LIN {X 0,Y 176.261,Z 619.953,A -85,B 0,C 180,E1 -22409.998,E2 -22409.998} C_VEL
LIN {X 0,Y 176.004,Z 621.002,A -85,B 0,C 180,E1 -22414.579,E2 -22414.579} C_VEL
LIN {X 0,Y 176.334,Z 620.73,A -85,B 0,C 180,E1 -22419.171,E2 -22419.171} C_VEL
LIN {X 0,Y 177.42,Z 619.155,A -85,B 0,C 180,E1 -22423.747,E2 -22423.747} C_VEL
LIN {X 0,Y 179.665,Z 616.268,A -85,B 0,C 180,E1 -22428.234,E2 -22428.234} C_VEL
LIN {X 0,Y 182.692,Z 611.986,A -85,B 0,C 180,E1 -22432.622,E2 -22432.622} C_VEL
LIN {X 0,Y 186.979,Z 606.194,A -85,B 0,C 180,E1 -22436.808,E2 -22436.808} C_VEL
LIN {X 0,Y 191.544,Z 599.723,A -85,B 0,C 180,E1 -22440.296,E2 -22440.296} C_VEL
LIN {X 0,Y 196.849,Z 591.739,A -85,B 0,C 180,E1 -22443.597,E2 -22443.597} C_VEL
LIN {X 0,Y 201.965,Z 583.426,A -85,B 0,C 180,E1 -22446.266,E2 -22446.266} C_VEL
LIN {X 0,Y 207.375,Z 573.579,A -85,B 0,C 180,E1 -22448.786,E2 -22448.786} C_VEL
LIN {X 0,Y 212.33,Z 563.502,A -85,B 0,C 180,E1 -22450.819,E2 -22450.819} C_VEL
LIN {X 0,Y 217.55,Z 551.5,A -85,B 0,C 180,E1 -22452.717,E2 -22452.717} C_VEL
LIN {X 0,Y 221.948,Z 539.683,A -85,B 0,C 180,E1 -22454.155,E2 -22454.155} C_VEL
LIN {X 0,Y 225.975,Z 526.726,A -85,B 0,C 180,E1 -22455.349,E2 -22455.349} C_VEL
LIN {X 0,Y 228.845,Z 514.868,A -85,B 0,C 180,E1 -22456.192,E2 -22456.192} C_VEL
LIN {X 0,Y 231.422,Z 500.809,A -85,B 0,C 180,E1 -22456.897,E2 -22456.897} C_VEL
LIN {X 0,Y 233.066,Z 485.237,A -85,B 0,C 180,E1 -22457.412,E2 -22457.412} C_VEL
LIN {X 0,Y 236.336,Z 441.448,A -85,B 0,C 180,E1 -22458.62,E2 -22458.62} C_VEL
LIN {X 0,Y 231.828,Z 430.629,A -85,B 0,C 180,E1 -22460.893,E2 -22460.893} C_VEL
LIN {X 0,Y 227.529,Z 421.656,A -85,B 0,C 180,E1 -22463.25,E2 -22463.25} C_VEL
LIN {X 0,Y 223.484,Z 413.857,A -85,B 0,C 180,E1 -22465.684,E2 -22465.684} C_VEL
LIN {X 0,Y 219.996,Z 407.651,A -85,B 0,C 180,E1 -22467.999,E2 -22467.999} C_VEL
LIN {X 0,Y 218.272,Z 404.689,A -85,B 0,C 180,E1 -22469.242,E2 -22469.242} C_VEL
LIN {X 0,Y 215.23,Z 399.598,A -85,B 0,C 180,E1 -22471.706,E2 -22471.706} C_VEL
LIN {X 0,Y 211.663,Z 393.98,A -85,B 0,C 180,E1 -22475.117,E2 -22475.117} C_VEL
LIN {X 0,Y 207.412,Z 387.519,A -85,B 0,C 180,E1 -22480.575,E2 -22480.575} C_VEL
LIN {X 0,Y 206.29,Z 386.531,A -85,B 0,C 180,E1 -22482.531,E2 -22482.531} C_VEL
LIN {X 0,Y 204.121,Z 383.562,A -85,B 0,C 180,E1 -22490.763,E2 -22490.763} C_VEL
LIN {X 0,Y 204.159,Z 383.555,A -85,B 0,C 180,E1 -22492.419,E2 -22492.419} C_VEL
LIN {X 0,Y 206.589,Z 386.339,A -85,B 0,C 180,E1 -22500.487,E2 -22500.487} C_VEL
LIN {X 0,Y 207.66,Z 387.333,A -85,B 0,C 180,E1 -22502.289,E2 -22502.289} C_VEL
LIN {X 0,Y 209.529,Z 390.505,A -85,B 0,C 180,E1 -22504.964,E2 -22504.964} C_VEL
LIN {X 0,Y 211.541,Z 392.569,A -85,B 0,C 180,E1 -22507.173,E2 -22507.173} C_VEL
LIN {X 0,Y 213.826,Z 396.048,A -85,B 0,C 180,E1 -22509.458,E2 -22509.458} C_VEL
LIN {X 0,Y 215.381,Z 397.913,A -85,B 0,C 180,E1 -22510.799,E2 -22510.799} C_VEL
LIN {X 0,Y 218.701,Z 402.698,A -85,B 0,C 180,E1 -22513.418,E2 -22513.418} C_VEL
LIN {X 0,Y 222.211,Z 407.786,A -85,B 0,C 180,E1 -22515.784,E2 -22515.784} C_VEL
LIN {X 0,Y 226.377,Z 414.067,A -85,B 0,C 180,E1 -22518.29,E2 -22518.29} C_VEL
LIN {X 0,Y 230.882,Z 421.436,A -85,B 0,C 180,E1 -22520.734,E2 -22520.734} C_VEL
LIN {X 0,Y 235.489,Z 429.755,A -85,B 0,C 180,E1 -22523.009,E2 -22523.009} C_VEL
LIN {X 0,Y 236.939,Z 432.896,A -85,B 0,C 180,E1 -22523.697,E2 -22523.697} C_VEL
LIN {X 0,Y 232.865,Z 484.514,A -85,B 0,C 180,E1 -22525.125,E2 -22525.125} C_VEL
LIN {X 0,Y 230.746,Z 498.985,A -85,B 0,C 180,E1 -22525.793,E2 -22525.793} C_VEL
LIN {X 0,Y 227.765,Z 513.123,A -85,B 0,C 180,E1 -22526.764,E2 -22526.764} C_VEL
LIN {X 0,Y 224.412,Z 525.3,A -85,B 0,C 180,E1 -22527.885,E2 -22527.885} C_VEL
LIN {X 0,Y 220.004,Z 538.449,A -85,B 0,C 180,E1 -22529.488,E2 -22529.488} C_VEL
LIN {X 0,Y 215.564,Z 549.31,A -85,B 0,C 180,E1 -22531.153,E2 -22531.153} C_VEL
LIN {X 0,Y 210.303,Z 560.524,A -85,B 0,C 180,E1 -22533.34,E2 -22533.34} C_VEL
LIN {X 0,Y 205.09,Z 570.271,A -85,B 0,C 180,E1 -22535.761,E2 -22535.761} C_VEL
LIN {X 0,Y 199.851,Z 579.024,A -85,B 0,C 180,E1 -22538.518,E2 -22538.518} C_VEL
LIN {X 0,Y 194.868,Z 586.574,A -85,B 0,C 180,E1 -22541.555,E2 -22541.555} C_VEL
LIN {X 0,Y 189.758,Z 593.653,A -85,B 0,C 180,E1 -22545.279,E2 -22545.279} C_VEL
LIN {X 0,Y 185.363,Z 599.272,A -85,B 0,C 180,E1 -22549.313,E2 -22549.313} C_VEL
LIN {X 0,Y 182.906,Z 602.168,A -85,B 0,C 180,E1 -22552.066,E2 -22552.066} C_VEL
LIN {X 0,Y 181.044,Z 604.278,A -85,B 0,C 180,E1 -22554.606,E2 -22554.606} C_VEL
LIN {X 0,Y 178.48,Z 606.841,A -85,B 0,C 180,E1 -22559.212,E2 -22559.212} C_VEL
LIN {X 0,Y 176.726,Z 607.981,A -85,B 0,C 180,E1 -22564.062,E2 -22564.062} C_VEL
LIN {X 0,Y 176.221,Z 607.996,A -85,B 0,C 180,E1 -22566.529,E2 -22566.529} C_VEL
LIN {X 0,Y 175.676,Z 606.957,A -85,B 0,C 180,E1 -22571.337,E2 -22571.337} C_VEL
LIN {X 0,Y 175.734,Z 605.894,A -85,B 0,C 180,E1 -22573.745,E2 -22573.745} C_VEL
LIN {X 0,Y 176.164,Z 602.698,A -85,B 0,C 180,E1 -22578.496,E2 -22578.496} C_VEL
LIN {X 0,Y 177.143,Z 598.549,A -85,B 0,C 180,E1 -22582.675,E2 -22582.675} C_VEL
LIN {X 0,Y 178.5,Z 593.339,A -85,B 0,C 180,E1 -22586.616,E2 -22586.616} C_VEL
LIN {X 0,Y 180.399,Z 586.664,A -85,B 0,C 180,E1 -22590.56,E2 -22590.56} C_VEL
LIN {X 0,Y 183.061,Z 578.344,A -85,B 0,C 180,E1 -22594.406,E2 -22594.406} C_VEL
LIN {X 0,Y 185.727,Z 569.663,A -85,B 0,C 180,E1 -22597.613,E2 -22597.613} C_VEL
LIN {X 0,Y 188.906,Z 559.128,A -85,B 0,C 180,E1 -22600.722,E2 -22600.722} C_VEL
LIN {X 0,Y 192.339,Z 547.305,A -85,B 0,C 180,E1 -22603.472,E2 -22603.472} C_VEL
LIN {X 0,Y 195.388,Z 535.469,A -85,B 0,C 180,E1 -22605.652,E2 -22605.652} C_VEL
LIN {X 0,Y 198.281,Z 522.429,A -85,B 0,C 180,E1 -22607.536,E2 -22607.536} C_VEL
LIN {X 0,Y 200.684,Z 509.152,A -85,B 0,C 180,E1 -22608.998,E2 -22608.998} C_VEL
LIN {X 0,Y 202.581,Z 494.605,A -85,B 0,C 180,E1 -22610.165,E2 -22610.165} C_VEL
LIN {X 0,Y 203.925,Z 480.192,A -85,B 0,C 180,E1 -22610.907,E2 -22610.907} C_VEL
LIN {X 0,Y 207.782,Z 410.461,A -85,B 0,C 180,E1 -22613.166,E2 -22613.166} C_VEL
LIN {X 0,Y 205.296,Z 404.053,A -85,B 0,C 180,E1 -22613.922,E2 -22613.922} C_VEL
LIN {X 0,Y 197.581,Z 388.625,A -85,B 0,C 180,E1 -22616.238,E2 -22616.238} C_VEL
LIN {X 0,Y 190.271,Z 375.852,A -85,B 0,C 180,E1 -22618.59,E2 -22618.59} C_VEL
LIN {X 0,Y 183.641,Z 365.472,A -85,B 0,C 180,E1 -22620.895,E2 -22620.895} C_VEL
LIN {X 0,Y 181.481,Z 362.093,A -85,B 0,C 180,E1 -22621.698,E2 -22621.698} C_VEL
LIN {X 0,Y 179.169,Z 359.175,A -85,B 0,C 180,E1 -22622.551,E2 -22622.551} C_VEL
LIN {X 0,Y 178.486,Z 356.878,A -85,B 0,C 180,E1 -22622.896,E2 -22622.896} C_VEL
LIN {X 0,Y 178.408,Z 356.871,A -85,B 0,C 180,E1 -22628.016,E2 -22628.016} C_VEL
LIN {X 0,Y 178.394,Z 356.874,A -85,B 0,C 180,E1 -22632.049,E2 -22632.049} C_VEL
LIN {X 0,Y 178.392,Z 356.857,A -85,B 0,C 180,E1 -22635.167,E2 -22635.167} C_VEL
LIN {X 0,Y 178.398,Z 356.885,A -85,B 0,C 180,E1 -22638.463,E2 -22638.463} C_VEL
LIN {X 0,Y 178.42,Z 356.842,A -85,B 0,C 180,E1 -22643.784,E2 -22643.784} C_VEL
LIN {X 0,Y 178.486,Z 356.856,A -85,B 0,C 180,E1 -22646.548,E2 -22646.548} C_VEL
LIN {X 0,Y 178.442,Z 356.873,A -85,B 0,C 180,E1 -22651.796,E2 -22651.796} C_VEL
LIN {X 0,Y 178.508,Z 356.875,A -85,B 0,C 180,E1 -22654.898,E2 -22654.898} C_VEL
LIN {X 0,Y 178.609,Z 356.861,A -85,B 0,C 180,E1 -22661.653,E2 -22661.653} C_VEL
LIN {X 0,Y 178.629,Z 356.813,A -85,B 0,C 180,E1 -22666.346,E2 -22666.346} C_VEL
LIN {X 0,Y 178.908,Z 356.807,A -85,B 0,C 180,E1 -22670.96,E2 -22670.96} C_VEL
LIN {X 0,Y 179.134,Z 356.761,A -85,B 0,C 180,E1 -22677.752,E2 -22677.752} C_VEL
LIN {X 0,Y 179.363,Z 356.721,A -85,B 0,C 180,E1 -22680.001,E2 -22680.001} C_VEL
LIN {X 0,Y 178.848,Z 356.83,A -85,B 0,C 180,E1 -22684.508,E2 -22684.508} C_VEL
LIN {X 0,Y 178.912,Z 356.815,A -85,B 0,C 180,E1 -22689.041,E2 -22689.041} C_VEL
LIN {X 0,Y 178.663,Z 356.846,A -85,B 0,C 180,E1 -22693.653,E2 -22693.653} C_VEL
LIN {X 0,Y 178.63,Z 356.847,A -85,B 0,C 180,E1 -22699.216,E2 -22699.216} C_VEL
LIN {X 0,Y 178.531,Z 356.859,A -85,B 0,C 180,E1 -22705.117,E2 -22705.117} C_VEL
LIN {X 0,Y 178.528,Z 356.862,A -85,B 0,C 180,E1 -22709.993,E2 -22709.993} C_VEL
LIN {X 0,Y 178.49,Z 356.872,A -85,B 0,C 180,E1 -22714.219,E2 -22714.219} C_VEL
LIN {X 0,Y 178.504,Z 356.951,A -85,B 0,C 180,E1 -22718.589,E2 -22718.589} C_VEL
LIN {X 0,Y 179.376,Z 359.579,A -85,B 0,C 180,E1 -22719.002,E2 -22719.002} C_VEL
LIN {X 0,Y 181.535,Z 362.296,A -85,B 0,C 180,E1 -22719.792,E2 -22719.792} C_VEL
LIN {X 0,Y 187.23,Z 372.234,A -85,B 0,C 180,E1 -22721.912,E2 -22721.912} C_VEL
LIN {X 0,Y 193.614,Z 385.014,A -85,B 0,C 180,E1 -22724.147,E2 -22724.147} C_VEL
LIN {X 0,Y 200.31,Z 400.306,A -85,B 0,C 180,E1 -22726.357,E2 -22726.357} C_VEL
LIN {X 0,Y 206.239,Z 416.491,A -85,B 0,C 180,E1 -22728.26,E2 -22728.26} C_VEL
LIN {X 0,Y 207.164,Z 425.712,A -85,B 0,C 180,E1 -22728.83,E2 -22728.83} C_VEL
LIN {X 0,Y 204.565,Z 475.041,A -85,B 0,C 180,E1 -22730.433,E2 -22730.433} C_VEL
LIN {X 0,Y 203.688,Z 480.877,A -85,B 0,C 180,E1 -22730.514,E2 -22730.514} C_VEL
LIN {X 0,Y 197.568,Z 499.736,A -85,B 0,C 180,E1 -22730.355,E2 -22730.355} C_VEL
LIN {X 0,Y 196.339,Z 505.475,A -85,B 0,C 180,E1 -22730.574,E2 -22730.574} C_VEL
LIN {X 0,Y 194.428,Z 518.993,A -85,B 0,C 180,E1 -22731.589,E2 -22731.589} C_VEL
LIN {X 0,Y 191.8,Z 532.414,A -85,B 0,C 180,E1 -22732.963,E2 -22732.963} C_VEL
LIN {X 0,Y 188.72,Z 545.437,A -85,B 0,C 180,E1 -22734.744,E2 -22734.744} C_VEL
LIN {X 0,Y 185.868,Z 556.719,A -85,B 0,C 180,E1 -22736.76,E2 -22736.76} C_VEL
LIN {X 0,Y 183.057,Z 566.038,A -85,B 0,C 180,E1 -22738.78,E2 -22738.78} C_VEL
LIN {X 0,Y 179.87,Z 575.945,A -85,B 0,C 180,E1 -22741.401,E2 -22741.401} C_VEL
LIN {X 0,Y 176.674,Z 585.85,A -85,B 0,C 180,E1 -22744.681,E2 -22744.681} C_VEL
LIN {X 0,Y 173.85,Z 594.782,A -85,B 0,C 180,E1 -22748.404,E2 -22748.404} C_VEL
LIN {X 0,Y 171.762,Z 601.876,A -85,B 0,C 180,E1 -22752.127,E2 -22752.127} C_VEL
LIN {X 0,Y 170.306,Z 607.294,A -85,B 0,C 180,E1 -22755.662,E2 -22755.662} C_VEL
LIN {X 0,Y 169.304,Z 612.981,A -85,B 0,C 180,E1 -22760.44,E2 -22760.44} C_VEL
LIN {X 0,Y 169.089,Z 615.207,A -85,B 0,C 180,E1 -22762.835,E2 -22762.835} C_VEL
LIN {X 0,Y 169.003,Z 617.786,A -85,B 0,C 180,E1 -22766.423,E2 -22766.423} C_VEL
LIN {X 0,Y 169.18,Z 619.597,A -85,B 0,C 180,E1 -22769.998,E2 -22769.998} C_VEL
LIN {X 0,Y 168.926,Z 620.714,A -85,B 0,C 180,E1 -22774.771,E2 -22774.771} C_VEL
LIN {X 0,Y 169.3,Z 620.515,A -85,B 0,C 180,E1 -22779.556,E2 -22779.556} C_VEL
LIN {X 0,Y 170.483,Z 619.019,A -85,B 0,C 180,E1 -22784.318,E2 -22784.318} C_VEL
LIN {X 0,Y 172.88,Z 616.212,A -85,B 0,C 180,E1 -22788.977,E2 -22788.977} C_VEL
LIN {X 0,Y 176.13,Z 612.015,A -85,B 0,C 180,E1 -22793.515,E2 -22793.515} C_VEL
LIN {X 0,Y 180.66,Z 606.311,A -85,B 0,C 180,E1 -22797.826,E2 -22797.826} C_VEL
LIN {X 0,Y 185.457,Z 599.935,A -85,B 0,C 180,E1 -22801.401,E2 -22801.401} C_VEL
LIN {X 0,Y 190.98,Z 592.059,A -85,B 0,C 180,E1 -22804.775,E2 -22804.775} C_VEL
LIN {X 0,Y 196.31,Z 583.865,A -85,B 0,C 180,E1 -22807.486,E2 -22807.486} C_VEL
LIN {X 0,Y 201.755,Z 574.456,A -85,B 0,C 180,E1 -22809.972,E2 -22809.972} C_VEL
LIN {X 0,Y 207.059,Z 564.249,A -85,B 0,C 180,E1 -22812.092,E2 -22812.092} C_VEL
LIN {X 0,Y 212.446,Z 552.457,A -85,B 0,C 180,E1 -22814.001,E2 -22814.001} C_VEL
LIN {X 0,Y 216.969,Z 540.917,A -85,B 0,C 180,E1 -22815.445,E2 -22815.445} C_VEL
LIN {X 0,Y 221.402,Z 527.401,A -85,B 0,C 180,E1 -22816.725,E2 -22816.725} C_VEL
LIN {X 0,Y 224.346,Z 515.777,A -85,B 0,C 180,E1 -22817.57,E2 -22817.57} C_VEL
LIN {X 0,Y 227.127,Z 501.604,A -85,B 0,C 180,E1 -22818.293,E2 -22818.293} C_VEL
LIN {X 0,Y 228.818,Z 486.854,A -85,B 0,C 180,E1 -22818.812,E2 -22818.812} C_VEL
LIN {X 0,Y 232.104,Z 444.116,A -85,B 0,C 180,E1 -22820.001,E2 -22820.001} C_VEL
LIN {X 0,Y 228.046,Z 434.201,A -85,B 0,C 180,E1 -22822.229,E2 -22822.229} C_VEL
LIN {X 0,Y 223.673,Z 424.769,A -85,B 0,C 180,E1 -22824.826,E2 -22824.826} C_VEL
LIN {X 0,Y 218.919,Z 415.596,A -85,B 0,C 180,E1 -22827.982,E2 -22827.982} C_VEL
LIN {X 0,Y 215.795,Z 410.218,A -85,B 0,C 180,E1 -22830.329,E2 -22830.329} C_VEL
LIN {X 0,Y 213.28,Z 405.755,A -85,B 0,C 180,E1 -22832.527,E2 -22832.527} C_VEL
LIN {X 0,Y 209.98,Z 400.378,A -85,B 0,C 180,E1 -22835.876,E2 -22835.876} C_VEL
LIN {X 0,Y 206.116,Z 394.154,A -85,B 0,C 180,E1 -22841.228,E2 -22841.228} C_VEL
LIN {X 0,Y 203.236,Z 390.606,A -85,B 0,C 180,E1 -22850.722,E2 -22850.722} C_VEL
LIN {X 0,Y 203.271,Z 390.593,A -85,B 0,C 180,E1 -22852.385,E2 -22852.385} C_VEL
LIN {X 0,Y 205.888,Z 393.57,A -85,B 0,C 180,E1 -22860.855,E2 -22860.855} C_VEL
LIN {X 0,Y 206.467,Z 394.216,A -85,B 0,C 180,E1 -22861.859,E2 -22861.859} C_VEL
LIN {X 0,Y 208.44,Z 397.561,A -85,B 0,C 180,E1 -22864.786,E2 -22864.786} C_VEL
LIN {X 0,Y 210.08,Z 399.305,A -85,B 0,C 180,E1 -22866.65,E2 -22866.65} C_VEL
LIN {X 0,Y 212.464,Z 402.895,A -85,B 0,C 180,E1 -22869.108,E2 -22869.108} C_VEL
LIN {X 0,Y 213.746,Z 404.582,A -85,B 0,C 180,E1 -22870.264,E2 -22870.264} C_VEL
LIN {X 0,Y 216.777,Z 409.088,A -85,B 0,C 180,E1 -22872.769,E2 -22872.769} C_VEL
LIN {X 0,Y 220.394,Z 414.504,A -85,B 0,C 180,E1 -22875.317,E2 -22875.317} C_VEL
LIN {X 0,Y 224.675,Z 421.287,A -85,B 0,C 180,E1 -22877.977,E2 -22877.977} C_VEL
LIN {X 0,Y 229.43,Z 429.452,A -85,B 0,C 180,E1 -22880.621,E2 -22880.621} C_VEL
LIN {X 0,Y 232.719,Z 435.879,A -85,B 0,C 180,E1 -22882.324,E2 -22882.324} C_VEL
LIN {X 0,Y 228.703,Z 485.113,A -85,B 0,C 180,E1 -22883.709,E2 -22883.709} C_VEL
LIN {X 0,Y 226.642,Z 498.883,A -85,B 0,C 180,E1 -22884.344,E2 -22884.344} C_VEL
LIN {X 0,Y 223.813,Z 512.028,A -85,B 0,C 180,E1 -22885.216,E2 -22885.216} C_VEL
LIN {X 0,Y 219.87,Z 526.017,A -85,B 0,C 180,E1 -22886.496,E2 -22886.496} C_VEL
LIN {X 0,Y 215.74,Z 537.951,A -85,B 0,C 180,E1 -22887.95,E2 -22887.95} C_VEL
LIN {X 0,Y 210.594,Z 550.126,A -85,B 0,C 180,E1 -22889.814,E2 -22889.814} C_VEL
LIN {X 0,Y 205.137,Z 561.245,A -85,B 0,C 180,E1 -22892.016,E2 -22892.016} C_VEL
LIN {X 0,Y 199.943,Z 570.521,A -85,B 0,C 180,E1 -22894.354,E2 -22894.354} C_VEL
LIN {X 0,Y 194.239,Z 579.602,A -85,B 0,C 180,E1 -22897.253,E2 -22897.253} C_VEL
LIN {X 0,Y 189.029,Z 587.098,A -85,B 0,C 180,E1 -22900.347,E2 -22900.347} C_VEL
LIN {X 0,Y 184.35,Z 593.206,A -85,B 0,C 180,E1 -22903.589,E2 -22903.589} C_VEL
LIN {X 0,Y 180.308,Z 598.131,A -85,B 0,C 180,E1 -22906.995,E2 -22906.995} C_VEL
LIN {X 0,Y 176.883,Z 602.005,A -85,B 0,C 180,E1 -22910.53,E2 -22910.53} C_VEL
LIN {X 0,Y 174.427,Z 604.602,A -85,B 0,C 180,E1 -22913.69,E2 -22913.69} C_VEL
LIN {X 0,Y 171.927,Z 606.907,A -85,B 0,C 180,E1 -22917.902,E2 -22917.902} C_VEL
LIN {X 0,Y 169.927,Z 608.23,A -85,B 0,C 180,E1 -22922.941,E2 -22922.941} C_VEL
LIN {X 0,Y 168.883,Z 608.039,A -85,B 0,C 180,E1 -22928.007,E2 -22928.007} C_VEL
LIN {X 0,Y 168.595,Z 606.409,A -85,B 0,C 180,E1 -22933.037,E2 -22933.037} C_VEL
LIN {X 0,Y 168.97,Z 603.345,A -85,B 0,C 180,E1 -22937.999,E2 -22937.999} C_VEL
LIN {X 0,Y 169.743,Z 600.065,A -85,B 0,C 180,E1 -22941.671,E2 -22941.671} C_VEL
LIN {X 0,Y 170.811,Z 595.914,A -85,B 0,C 180,E1 -22945.282,E2 -22945.282} C_VEL
LIN {X 0,Y 172.279,Z 590.738,A -85,B 0,C 180,E1 -22948.833,E2 -22948.833} C_VEL
LIN {X 0,Y 174.641,Z 583.348,A -85,B 0,C 180,E1 -22952.885,E2 -22952.885} C_VEL
LIN {X 0,Y 177.738,Z 574.158,A -85,B 0,C 180,E1 -22956.815,E2 -22956.815} C_VEL
LIN {X 0,Y 180.753,Z 564.552,A -85,B 0,C 180,E1 -22960.079,E2 -22960.079} C_VEL
LIN {X 0,Y 184.07,Z 553.872,A -85,B 0,C 180,E1 -22962.964,E2 -22962.964} C_VEL
LIN {X 0,Y 187.427,Z 542.056,A -85,B 0,C 180,E1 -22965.498,E2 -22965.498} C_VEL
LIN {X 0,Y 190.738,Z 528.898,A -85,B 0,C 180,E1 -22967.699,E2 -22967.699} C_VEL
LIN {X 0,Y 193.347,Z 516.33,A -85,B 0,C 180,E1 -22969.324,E2 -22969.324} C_VEL
LIN {X 0,Y 195.596,Z 502.567,A -85,B 0,C 180,E1 -22970.666,E2 -22970.666} C_VEL
LIN {X 0,Y 197.296,Z 488.463,A -85,B 0,C 180,E1 -22971.618,E2 -22971.618} C_VEL
LIN {X 0,Y 198.522,Z 472.121,A -85,B 0,C 180,E1 -22972.282,E2 -22972.282} C_VEL
LIN {X 0,Y 201.874,Z 411.942,A -85,B 0,C 180,E1 -22974.264,E2 -22974.264} C_VEL
LIN {X 0,Y 196.905,Z 400.974,A -85,B 0,C 180,E1 -22975.814,E2 -22975.814} C_VEL
LIN {X 0,Y 189.681,Z 387.165,A -85,B 0,C 180,E1 -22978.174,E2 -22978.174} C_VEL
LIN {X 0,Y 183.223,Z 376.303,A -85,B 0,C 180,E1 -22980.439,E2 -22980.439} C_VEL
LIN {X 0,Y 179.128,Z 370.041,A -85,B 0,C 180,E1 -22981.961,E2 -22981.961} C_VEL
LIN {X 0,Y 176.415,Z 366.014,A -85,B 0,C 180,E1 -22983.022,E2 -22983.022} C_VEL
LIN {X 0,Y 174.06,Z 362.431,A -85,B 0,C 180,E1 -22983.985,E2 -22983.985} C_VEL
LIN {X 0,Y 172.1,Z 360.028,A -85,B 0,C 180,E1 -22984.785,E2 -22984.785} C_VEL
LIN {X 0,Y 171.39,Z 357.744,A -85,B 0,C 180,E1 -22985.239,E2 -22985.239} C_VEL
LIN {X 0,Y 171.344,Z 357.758,A -85,B 0,C 180,E1 -22988.803,E2 -22988.803} C_VEL
LIN {X 0,Y 171.319,Z 357.735,A -85,B 0,C 180,E1 -22994.22,E2 -22994.22} C_VEL
LIN {X 0,Y 171.331,Z 357.766,A -85,B 0,C 180,E1 -22998.981,E2 -22998.981} C_VEL
LIN {X 0,Y 171.361,Z 357.731,A -85,B 0,C 180,E1 -23002.035,E2 -23002.035} C_VEL
LIN {X 0,Y 171.4,Z 357.719,A -85,B 0,C 180,E1 -23005.095,E2 -23005.095} C_VEL
LIN {X 0,Y 171.41,Z 357.755,A -85,B 0,C 180,E1 -23010.528,E2 -23010.528} C_VEL
LIN {X 0,Y 171.43,Z 357.756,A -85,B 0,C 180,E1 -23015.798,E2 -23015.798} C_VEL
LIN {X 0,Y 171.511,Z 357.745,A -85,B 0,C 180,E1 -23020.865,E2 -23020.865} C_VEL
LIN {X 0,Y 171.545,Z 357.699,A -85,B 0,C 180,E1 -23025.771,E2 -23025.771} C_VEL
LIN {X 0,Y 171.847,Z 357.682,A -85,B 0,C 180,E1 -23030.586,E2 -23030.586} C_VEL
LIN {X 0,Y 171.796,Z 357.702,A -85,B 0,C 180,E1 -23035.308,E2 -23035.308} C_VEL
LIN {X 0,Y 172.327,Z 357.596,A -85,B 0,C 180,E1 -23040.001,E2 -23040.001} C_VEL
LIN {X 0,Y 171.868,Z 357.696,A -85,B 0,C 180,E1 -23047.047,E2 -23047.047} C_VEL
LIN {X 0,Y 171.774,Z 357.713,A -85,B 0,C 180,E1 -23050.897,E2 -23050.897} C_VEL
LIN {X 0,Y 171.56,Z 357.74,A -85,B 0,C 180,E1 -23056.665,E2 -23056.665} C_VEL
LIN {X 0,Y 171.551,Z 357.727,A -85,B 0,C 180,E1 -23059.562,E2 -23059.562} C_VEL
LIN {X 0,Y 171.468,Z 357.739,A -85,B 0,C 180,E1 -23065.611,E2 -23065.611} C_VEL
LIN {X 0,Y 171.446,Z 357.746,A -85,B 0,C 180,E1 -23070.585,E2 -23070.585} C_VEL
LIN {X 0,Y 171.381,Z 357.753,A -85,B 0,C 180,E1 -23076.304,E2 -23076.304} C_VEL
LIN {X 0,Y 172.335,Z 360.479,A -85,B 0,C 180,E1 -23076.797,E2 -23076.797} C_VEL
LIN {X 0,Y 174.274,Z 362.579,A -85,B 0,C 180,E1 -23077.568,E2 -23077.568} C_VEL
LIN {X 0,Y 176.733,Z 366.484,A -85,B 0,C 180,E1 -23078.577,E2 -23078.577} C_VEL
LIN {X 0,Y 181.064,Z 373.766,A -85,B 0,C 180,E1 -23080.28,E2 -23080.28} C_VEL
LIN {X 0,Y 185.126,Z 381.484,A -85,B 0,C 180,E1 -23081.826,E2 -23081.826} C_VEL
LIN {X 0,Y 191.167,Z 394.289,A -85,B 0,C 180,E1 -23084.009,E2 -23084.009} C_VEL
LIN {X 0,Y 196.682,Z 407.982,A -85,B 0,C 180,E1 -23085.925,E2 -23085.925} C_VEL
LIN {X 0,Y 200.633,Z 419.431,A -85,B 0,C 180,E1 -23087.279,E2 -23087.279} C_VEL
LIN {X 0,Y 201.287,Z 426.847,A -85,B 0,C 180,E1 -23087.738,E2 -23087.738} C_VEL
LIN {X 0,Y 197.341,Z 496.005,A -85,B 0,C 180,E1 -23090.067,E2 -23090.067} C_VEL
LIN {X 0,Y 196.339,Z 505.475,A -85,B 0,C 180,E1 -23090.574,E2 -23090.574} C_VEL
LIN {X 0,Y 194.333,Z 513.011,A -85,B 0,C 180,E1 -23090.909,E2 -23090.909} C_VEL
LIN {X 0,Y 187.752,Z 527.343,A -85,B 0,C 180,E1 -23091.486,E2 -23091.486} C_VEL
LIN {X 0,Y 185.679,Z 532.688,A -85,B 0,C 180,E1 -23091.944,E2 -23091.944} C_VEL
LIN {X 0,Y 185.166,Z 534.474,A -85,B 0,C 180,E1 -23092.15,E2 -23092.15} C_VEL
LIN {X 0,Y 182.128,Z 546.755,A -85,B 0,C 180,E1 -23093.949,E2 -23093.949} C_VEL
LIN {X 0,Y 179.392,Z 556.978,A -85,B 0,C 180,E1 -23095.859,E2 -23095.859} C_VEL
LIN {X 0,Y 176.285,Z 566.899,A -85,B 0,C 180,E1 -23098.111,E2 -23098.111} C_VEL
LIN {X 0,Y 172.959,Z 576.61,A -85,B 0,C 180,E1 -23100.814,E2 -23100.814} C_VEL
LIN {X 0,Y 169.711,Z 586.367,A -85,B 0,C 180,E1 -23104.224,E2 -23104.224} C_VEL
LIN {X 0,Y 166.975,Z 594.584,A -85,B 0,C 180,E1 -23107.819,E2 -23107.819} C_VEL
LIN {X 0,Y 164.936,Z 601.113,A -85,B 0,C 180,E1 -23111.36,E2 -23111.36} C_VEL
LIN {X 0,Y 163.379,Z 606.634,A -85,B 0,C 180,E1 -23115.041,E2 -23115.041} C_VEL
LIN {X 0,Y 162.278,Z 612.416,A -85,B 0,C 180,E1 -23120.022,E2 -23120.022} C_VEL
LIN {X 0,Y 161.923,Z 616.563,A -85,B 0,C 180,E1 -23125.018,E2 -23125.018} C_VEL
LIN {X 0,Y 162.081,Z 619.212,A -85,B 0,C 180,E1 -23129.998,E2 -23129.998} C_VEL
LIN {X 0,Y 161.875,Z 620.092,A -85,B 0,C 180,E1 -23133.046,E2 -23133.046} C_VEL
LIN {X 0,Y 161.932,Z 620.52,A -85,B 0,C 180,E1 -23137.479,E2 -23137.479} C_VEL
LIN {X 0,Y 162.792,Z 619.752,A -85,B 0,C 180,E1 -23142.463,E2 -23142.463} C_VEL
LIN {X 0,Y 164.735,Z 617.687,A -85,B 0,C 180,E1 -23147.373,E2 -23147.373} C_VEL
LIN {X 0,Y 167.769,Z 614.279,A -85,B 0,C 180,E1 -23152.147,E2 -23152.147} C_VEL
LIN {X 0,Y 170.735,Z 610.789,A -85,B 0,C 180,E1 -23155.606,E2 -23155.606} C_VEL
LIN {X 0,Y 175.732,Z 604.806,A -85,B 0,C 180,E1 -23159.991,E2 -23159.991} C_VEL
LIN {X 0,Y 181.012,Z 598.127,A -85,B 0,C 180,E1 -23163.589,E2 -23163.589} C_VEL
LIN {X 0,Y 186.994,Z 589.871,A -85,B 0,C 180,E1 -23166.964,E2 -23166.964} C_VEL
LIN {X 0,Y 192.667,Z 581.309,A -85,B 0,C 180,E1 -23169.666,E2 -23169.666} C_VEL
LIN {X 0,Y 198.643,Z 570.995,A -85,B 0,C 180,E1 -23172.236,E2 -23172.236} C_VEL
LIN {X 0,Y 204.606,Z 559.496,A -85,B 0,C 180,E1 -23174.413,E2 -23174.413} C_VEL
LIN {X 0,Y 210.286,Z 546.656,A -85,B 0,C 180,E1 -23176.278,E2 -23176.278} C_VEL
LIN {X 0,Y 215.123,Z 533.815,A -85,B 0,C 180,E1 -23177.656,E2 -23177.656} C_VEL
LIN {X 0,Y 219.033,Z 520.545,A -85,B 0,C 180,E1 -23178.763,E2 -23178.763} C_VEL
LIN {X 0,Y 222.357,Z 506.015,A -85,B 0,C 180,E1 -23179.582,E2 -23179.582} C_VEL
LIN {X 0,Y 224.435,Z 491.745,A -85,B 0,C 180,E1 -23180.152,E2 -23180.152} C_VEL
LIN {X 0,Y 228.089,Z 446.972,A -85,B 0,C 180,E1 -23181.423,E2 -23181.423} C_VEL
LIN {X 0,Y 224.238,Z 437.385,A -85,B 0,C 180,E1 -23183.706,E2 -23183.706} C_VEL
LIN {X 0,Y 220.009,Z 428.358,A -85,B 0,C 180,E1 -23186.412,E2 -23186.412} C_VEL
LIN {X 0,Y 216.252,Z 420.862,A -85,B 0,C 180,E1 -23189.114,E2 -23189.114} C_VEL
LIN {X 0,Y 213.558,Z 415.935,A -85,B 0,C 180,E1 -23191.326,E2 -23191.326} C_VEL
LIN {X 0,Y 211.529,Z 412.129,A -85,B 0,C 180,E1 -23193.216,E2 -23193.216} C_VEL
LIN {X 0,Y 208.465,Z 406.932,A -85,B 0,C 180,E1 -23196.499,E2 -23196.499} C_VEL
LIN {X 0,Y 204.905,Z 400.932,A -85,B 0,C 180,E1 -23201.761,E2 -23201.761} C_VEL
LIN {X 0,Y 202.345,Z 397.667,A -85,B 0,C 180,E1 -23210.681,E2 -23210.681} C_VEL
LIN {X 0,Y 202.372,Z 397.669,A -85,B 0,C 180,E1 -23212.351,E2 -23212.351} C_VEL
LIN {X 0,Y 204.519,Z 400.262,A -85,B 0,C 180,E1 -23219.999,E2 -23219.999} C_VEL
LIN {X 0,Y 205.322,Z 401.215,A -85,B 0,C 180,E1 -23221.501,E2 -23221.501} C_VEL
LIN {X 0,Y 207.195,Z 404.412,A -85,B 0,C 180,E1 -23224.406,E2 -23224.406} C_VEL
LIN {X 0,Y 208.688,Z 406.089,A -85,B 0,C 180,E1 -23226.175,E2 -23226.175} C_VEL
LIN {X 0,Y 211.107,Z 409.755,A -85,B 0,C 180,E1 -23228.752,E2 -23228.752} C_VEL
LIN {X 0,Y 214.459,Z 414.715,A -85,B 0,C 180,E1 -23231.744,E2 -23231.744} C_VEL
LIN {X 0,Y 219.285,Z 422.243,A -85,B 0,C 180,E1 -23235.304,E2 -23235.304} C_VEL
LIN {X 0,Y 224.718,Z 431.483,A -85,B 0,C 180,E1 -23238.684,E2 -23238.684} C_VEL
LIN {X 0,Y 228.68,Z 438.964,A -85,B 0,C 180,E1 -23240.893,E2 -23240.893} C_VEL
LIN {X 0,Y 224.754,Z 485.669,A -85,B 0,C 180,E1 -23242.233,E2 -23242.233} C_VEL
LIN {X 0,Y 222.631,Z 499.216,A -85,B 0,C 180,E1 -23242.853,E2 -23242.853} C_VEL
LIN {X 0,Y 219.404,Z 513.468,A -85,B 0,C 180,E1 -23243.811,E2 -23243.811} C_VEL
LIN {X 0,Y 215.275,Z 527.368,A -85,B 0,C 180,E1 -23245.112,E2 -23245.112} C_VEL
LIN {X 0,Y 211.093,Z 538.81,A -85,B 0,C 180,E1 -23246.527,E2 -23246.527} C_VEL
LIN {X 0,Y 205.661,Z 551.119,A -85,B 0,C 180,E1 -23248.442,E2 -23248.442} C_VEL
LIN {X 0,Y 200.079,Z 561.963,A -85,B 0,C 180,E1 -23250.622,E2 -23250.622} C_VEL
LIN {X 0,Y 194.927,Z 570.766,A -85,B 0,C 180,E1 -23252.873,E2 -23252.873} C_VEL
LIN {X 0,Y 188.818,Z 580.047,A -85,B 0,C 180,E1 -23255.87,E2 -23255.87} C_VEL
LIN {X 0,Y 183.271,Z 587.612,A -85,B 0,C 180,E1 -23259.059,E2 -23259.059} C_VEL
LIN {X 0,Y 177.556,Z 594.598,A -85,B 0,C 180,E1 -23262.964,E2 -23262.964} C_VEL
LIN {X 0,Y 172.805,Z 599.95,A -85,B 0,C 180,E1 -23267.058,E2 -23267.058} C_VEL
LIN {X 0,Y 168.878,Z 603.952,A -85,B 0,C 180,E1 -23271.377,E2 -23271.377} C_VEL
LIN {X 0,Y 165.474,Z 606.958,A -85,B 0,C 180,E1 -23276.489,E2 -23276.489} C_VEL
LIN {X 0,Y 163.17,Z 608.428,A -85,B 0,C 180,E1 -23281.722,E2 -23281.722} C_VEL
LIN {X 0,Y 161.919,Z 608.414,A -85,B 0,C 180,E1 -23287.008,E2 -23287.008} C_VEL
LIN {X 0,Y 161.491,Z 606.918,A -85,B 0,C 180,E1 -23292.266,E2 -23292.266} C_VEL
LIN {X 0,Y 161.559,Z 605.629,A -85,B 0,C 180,E1 -23294.873,E2 -23294.873} C_VEL
LIN {X 0,Y 162.27,Z 601.955,A -85,B 0,C 180,E1 -23300.026,E2 -23300.026} C_VEL
LIN {X 0,Y 163.264,Z 598.092,A -85,B 0,C 180,E1 -23303.927,E2 -23303.927} C_VEL
LIN {X 0,Y 164.559,Z 593.533,A -85,B 0,C 180,E1 -23307.554,E2 -23307.554} C_VEL
LIN {X 0,Y 166.722,Z 586.758,A -85,B 0,C 180,E1 -23311.814,E2 -23311.814} C_VEL
LIN {X 0,Y 169.538,Z 578.638,A -85,B 0,C 180,E1 -23315.802,E2 -23315.802} C_VEL
LIN {X 0,Y 172.592,Z 569.496,A -85,B 0,C 180,E1 -23319.376,E2 -23319.376} C_VEL
LIN {X 0,Y 176.131,Z 558.805,A -85,B 0,C 180,E1 -23322.679,E2 -23322.679} C_VEL
LIN {X 0,Y 179.503,Z 547.994,A -85,B 0,C 180,E1 -23325.326,E2 -23325.326} C_VEL
LIN {X 0,Y 182.832,Z 536.169,A -85,B 0,C 180,E1 -23327.623,E2 -23327.623} C_VEL
LIN {X 0,Y 185.918,Z 523.174,A -85,B 0,C 180,E1 -23329.604,E2 -23329.604} C_VEL
LIN {X 0,Y 188.615,Z 509.378,A -85,B 0,C 180,E1 -23331.19,E2 -23331.19} C_VEL
LIN {X 0,Y 190.592,Z 495.475,A -85,B 0,C 180,E1 -23332.352,E2 -23332.352} C_VEL
LIN {X 0,Y 191.977,Z 481.85,A -85,B 0,C 180,E1 -23333.106,E2 -23333.106} C_VEL
LIN {X 0,Y 196.039,Z 414.514,A -85,B 0,C 180,E1 -23335.379,E2 -23335.379} C_VEL
LIN {X 0,Y 195.436,Z 412.406,A -85,B 0,C 180,E1 -23335.609,E2 -23335.609} C_VEL
LIN {X 0,Y 188.166,Z 397.333,A -85,B 0,C 180,E1 -23338.046,E2 -23338.046} C_VEL
LIN {X 0,Y 181.361,Z 385.035,A -85,B 0,C 180,E1 -23340.497,E2 -23340.497} C_VEL
LIN {X 0,Y 175.189,Z 375.186,A -85,B 0,C 180,E1 -23342.883,E2 -23342.883} C_VEL
LIN {X 0,Y 171.991,Z 370.517,A -85,B 0,C 180,E1 -23344.192,E2 -23344.192} C_VEL
LIN {X 0,Y 170.197,Z 367.779,A -85,B 0,C 180,E1 -23344.966,E2 -23344.966} C_VEL
LIN {X 0,Y 168,Z 364.707,A -85,B 0,C 180,E1 -23345.935,E2 -23345.935} C_VEL
LIN {X 0,Y 167.175,Z 363.442,A -85,B 0,C 180,E1 -23346.317,E2 -23346.317} C_VEL
LIN {X 0,Y 165.255,Z 361.357,A -85,B 0,C 180,E1 -23347.176,E2 -23347.176} C_VEL
LIN {X 0,Y 164.323,Z 358.621,A -85,B 0,C 180,E1 -23347.778,E2 -23347.778} C_VEL
LIN {X 0,Y 164.281,Z 358.614,A -85,B 0,C 180,E1 -23353.344,E2 -23353.344} C_VEL
LIN {X 0,Y 164.261,Z 358.63,A -85,B 0,C 180,E1 -23356.8,E2 -23356.8} C_VEL
LIN {X 0,Y 164.291,Z 358.635,A -85,B 0,C 180,E1 -23360.357,E2 -23360.357} C_VEL
LIN {X 0,Y 164.328,Z 358.594,A -85,B 0,C 180,E1 -23364.353,E2 -23364.353} C_VEL
LIN {X 0,Y 164.373,Z 358.635,A -85,B 0,C 180,E1 -23369.132,E2 -23369.132} C_VEL
LIN {X 0,Y 164.389,Z 358.633,A -85,B 0,C 180,E1 -23374.691,E2 -23374.691} C_VEL
LIN {X 0,Y 164.42,Z 358.624,A -85,B 0,C 180,E1 -23380.119,E2 -23380.119} C_VEL
LIN {X 0,Y 164.475,Z 358.585,A -85,B 0,C 180,E1 -23385.146,E2 -23385.146} C_VEL
LIN {X 0,Y 164.767,Z 358.554,A -85,B 0,C 180,E1 -23390.177,E2 -23390.177} C_VEL
LIN {X 0,Y 164.825,Z 358.575,A -85,B 0,C 180,E1 -23392.652,E2 -23392.652} C_VEL
LIN {X 0,Y 165.29,Z 358.47,A -85,B 0,C 180,E1 -23400.001,E2 -23400.001} C_VEL
LIN {X 0,Y 164.829,Z 358.57,A -85,B 0,C 180,E1 -23407.35,E2 -23407.35} C_VEL
LIN {X 0,Y 164.708,Z 358.593,A -85,B 0,C 180,E1 -23411.06,E2 -23411.06} C_VEL
LIN {X 0,Y 164.49,Z 358.618,A -85,B 0,C 180,E1 -23417.403,E2 -23417.403} C_VEL
LIN {X 0,Y 164.48,Z 358.608,A -85,B 0,C 180,E1 -23419.989,E2 -23419.989} C_VEL
LIN {X 0,Y 164.394,Z 358.622,A -85,B 0,C 180,E1 -23426.13,E2 -23426.13} C_VEL
LIN {X 0,Y 164.384,Z 358.63,A -85,B 0,C 180,E1 -23432.374,E2 -23432.374} C_VEL
LIN {X 0,Y 164.366,Z 358.827,A -85,B 0,C 180,E1 -23433.771,E2 -23433.771} C_VEL
LIN {X 0,Y 165.263,Z 361.329,A -85,B 0,C 180,E1 -23434.287,E2 -23434.287} C_VEL
LIN {X 0,Y 167.323,Z 363.574,A -85,B 0,C 180,E1 -23435.211,E2 -23435.211} C_VEL
LIN {X 0,Y 169.918,Z 367.53,A -85,B 0,C 180,E1 -23436.39,E2 -23436.39} C_VEL
LIN {X 0,Y 171.405,Z 369.637,A -85,B 0,C 180,E1 -23437.03,E2 -23437.03} C_VEL
LIN {X 0,Y 174.72,Z 374.683,A -85,B 0,C 180,E1 -23438.412,E2 -23438.412} C_VEL
LIN {X 0,Y 180.319,Z 385.245,A -85,B 0,C 180,E1 -23440.688,E2 -23440.688} C_VEL
LIN {X 0,Y 186.375,Z 398.383,A -85,B 0,C 180,E1 -23443.021,E2 -23443.021} C_VEL
LIN {X 0,Y 191.688,Z 411.962,A -85,B 0,C 180,E1 -23444.986,E2 -23444.986} C_VEL
LIN {X 0,Y 195.002,Z 421.512,A -85,B 0,C 180,E1 -23446.183,E2 -23446.183} C_VEL
LIN {X 0,Y 195.461,Z 427.757,A -85,B 0,C 180,E1 -23446.57,E2 -23446.57} C_VEL
LIN {X 0,Y 191.441,Z 495.576,A -85,B 0,C 180,E1 -23448.899,E2 -23448.899} C_VEL
LIN {X 0,Y 189.836,Z 509.459,A -85,B 0,C 180,E1 -23449.703,E2 -23449.703} C_VEL
LIN {X 0,Y 187.503,Z 523.711,A -85,B 0,C 180,E1 -23450.935,E2 -23450.935} C_VEL
LIN {X 0,Y 185.166,Z 534.474,A -85,B 0,C 180,E1 -23452.15,E2 -23452.15} C_VEL
LIN {X 0,Y 183.285,Z 539.763,A -85,B 0,C 180,E1 -23452.754,E2 -23452.754} C_VEL
LIN {X 0,Y 178.721,Z 548.035,A -85,B 0,C 180,E1 -23453.657,E2 -23453.657} C_VEL
LIN {X 0,Y 173.943,Z 556.053,A -85,B 0,C 180,E1 -23454.756,E2 -23454.756} C_VEL
LIN {X 0,Y 171.756,Z 560.755,A -85,B 0,C 180,E1 -23455.665,E2 -23455.665} C_VEL
LIN {X 0,Y 168.098,Z 571.736,A -85,B 0,C 180,E1 -23458.49,E2 -23458.49} C_VEL
LIN {X 0,Y 164.332,Z 582.311,A -85,B 0,C 180,E1 -23461.935,E2 -23461.935} C_VEL
LIN {X 0,Y 161.299,Z 591.03,A -85,B 0,C 180,E1 -23465.546,E2 -23465.546} C_VEL
LIN {X 0,Y 158.519,Z 599.324,A -85,B 0,C 180,E1 -23469.901,E2 -23469.901} C_VEL
LIN {X 0,Y 156.477,Z 605.97,A -85,B 0,C 180,E1 -23474.364,E2 -23474.364} C_VEL
LIN {X 0,Y 155.232,Z 611.842,A -85,B 0,C 180,E1 -23479.564,E2 -23479.564} C_VEL
LIN {X 0,Y 154.841,Z 616.077,A -85,B 0,C 180,E1 -23484.789,E2 -23484.789} C_VEL
LIN {X 0,Y 154.986,Z 618.808,A -85,B 0,C 180,E1 -23489.998,E2 -23489.998} C_VEL
LIN {X 0,Y 154.815,Z 619.702,A -85,B 0,C 180,E1 -23492.892,E2 -23492.892} C_VEL
LIN {X 0,Y 154.887,Z 620.238,A -85,B 0,C 180,E1 -23497.821,E2 -23497.821} C_VEL
LIN {X 0,Y 155.828,Z 619.553,A -85,B 0,C 180,E1 -23503.03,E2 -23503.03} C_VEL
LIN {X 0,Y 157.93,Z 617.577,A -85,B 0,C 180,E1 -23508.147,E2 -23508.147} C_VEL
LIN {X 0,Y 161.157,Z 614.263,A -85,B 0,C 180,E1 -23513.107,E2 -23513.107} C_VEL
LIN {X 0,Y 165.546,Z 609.504,A -85,B 0,C 180,E1 -23517.836,E2 -23517.836} C_VEL
LIN {X 0,Y 171.083,Z 603.172,A -85,B 0,C 180,E1 -23522.276,E2 -23522.276} C_VEL
LIN {X 0,Y 176.803,Z 596.175,A -85,B 0,C 180,E1 -23525.893,E2 -23525.893} C_VEL
LIN {X 0,Y 183.296,Z 587.551,A -85,B 0,C 180,E1 -23529.243,E2 -23529.243} C_VEL
LIN {X 0,Y 189.253,Z 578.601,A -85,B 0,C 180,E1 -23531.944,E2 -23531.944} C_VEL
LIN {X 0,Y 194.572,Z 569.757,A -85,B 0,C 180,E1 -23534.049,E2 -23534.049} C_VEL
LIN {X 0,Y 200.815,Z 558.089,A -85,B 0,C 180,E1 -23536.202,E2 -23536.202} C_VEL
LIN {X 0,Y 206.111,Z 546.448,A -85,B 0,C 180,E1 -23537.868,E2 -23537.868} C_VEL
LIN {X 0,Y 211.09,Z 533.631,A -85,B 0,C 180,E1 -23539.235,E2 -23539.235} C_VEL
LIN {X 0,Y 215.125,Z 520.383,A -85,B 0,C 180,E1 -23540.33,E2 -23540.33} C_VEL
LIN {X 0,Y 218.484,Z 506.193,A -85,B 0,C 180,E1 -23541.128,E2 -23541.128} C_VEL
LIN {X 0,Y 220.687,Z 491.622,A -85,B 0,C 180,E1 -23541.709,E2 -23541.709} C_VEL
LIN {X 0,Y 224.23,Z 449.931,A -85,B 0,C 180,E1 -23542.887,E2 -23542.887} C_VEL
LIN {X 0,Y 220.244,Z 439.918,A -85,B 0,C 180,E1 -23545.449,E2 -23545.449} C_VEL
LIN {X 0,Y 216.153,Z 431.103,A -85,B 0,C 180,E1 -23548.331,E2 -23548.331} C_VEL
LIN {X 0,Y 213.068,Z 424.742,A -85,B 0,C 180,E1 -23550.835,E2 -23550.835} C_VEL
LIN {X 0,Y 209.77,Z 418.467,A -85,B 0,C 180,E1 -23553.954,E2 -23553.954} C_VEL
LIN {X 0,Y 206.911,Z 413.411,A -85,B 0,C 180,E1 -23557.207,E2 -23557.207} C_VEL
LIN {X 0,Y 203.902,Z 407.945,A -85,B 0,C 180,E1 -23561.928,E2 -23561.928} C_VEL
LIN {X 0,Y 201.452,Z 404.733,A -85,B 0,C 180,E1 -23570.639,E2 -23570.639} C_VEL
LIN {X 0,Y 201.474,Z 404.731,A -85,B 0,C 180,E1 -23572.317,E2 -23572.317} C_VEL
LIN {X 0,Y 203.808,Z 407.502,A -85,B 0,C 180,E1 -23580.376,E2 -23580.376} C_VEL
LIN {X 0,Y 204.517,Z 408.946,A -85,B 0,C 180,E1 -23581.784,E2 -23581.784} C_VEL
LIN {X 0,Y 207.336,Z 412.971,A -85,B 0,C 180,E1 -23585.733,E2 -23585.733} C_VEL
LIN {X 0,Y 210.358,Z 417.576,A -85,B 0,C 180,E1 -23588.992,E2 -23588.992} C_VEL
LIN {X 0,Y 213.54,Z 422.721,A -85,B 0,C 180,E1 -23591.859,E2 -23591.859} C_VEL
LIN {X 0,Y 217.13,Z 428.471,A -85,B 0,C 180,E1 -23594.588,E2 -23594.588} C_VEL
LIN {X 0,Y 222.247,Z 437.469,A -85,B 0,C 180,E1 -23597.926,E2 -23597.926} C_VEL
LIN {X 0,Y 224.807,Z 442.391,A -85,B 0,C 180,E1 -23599.442,E2 -23599.442} C_VEL
LIN {X 0,Y 221.046,Z 485.613,A -85,B 0,C 180,E1 -23600.676,E2 -23600.676} C_VEL
LIN {X 0,Y 218.951,Z 498.807,A -85,B 0,C 180,E1 -23601.263,E2 -23601.263} C_VEL
LIN {X 0,Y 215.802,Z 512.608,A -85,B 0,C 180,E1 -23602.168,E2 -23602.168} C_VEL
LIN {X 0,Y 212.01,Z 525.322,A -85,B 0,C 180,E1 -23603.304,E2 -23603.304} C_VEL
LIN {X 0,Y 207.203,Z 538.37,A -85,B 0,C 180,E1 -23604.868,E2 -23604.868} C_VEL
LIN {X 0,Y 201.7,Z 550.476,A -85,B 0,C 180,E1 -23606.712,E2 -23606.712} C_VEL
LIN {X 0,Y 195.746,Z 561.704,A -85,B 0,C 180,E1 -23608.942,E2 -23608.942} C_VEL
LIN {X 0,Y 189.593,Z 571.741,A -85,B 0,C 180,E1 -23611.511,E2 -23611.511} C_VEL
LIN {X 0,Y 183.326,Z 580.725,A -85,B 0,C 180,E1 -23614.494,E2 -23614.494} C_VEL
LIN {X 0,Y 177.6,Z 588.115,A -85,B 0,C 180,E1 -23617.683,E2 -23617.683} C_VEL
LIN {X 0,Y 172.079,Z 594.551,A -85,B 0,C 180,E1 -23621.332,E2 -23621.332} C_VEL
LIN {X 0,Y 166.684,Z 600.265,A -85,B 0,C 180,E1 -23625.788,E2 -23625.788} C_VEL
LIN {X 0,Y 162.924,Z 603.862,A -85,B 0,C 180,E1 -23629.684,E2 -23629.684} C_VEL
LIN {X 0,Y 160.882,Z 605.634,A -85,B 0,C 180,E1 -23632.299,E2 -23632.299} C_VEL
LIN {X 0,Y 157.692,Z 607.998,A -85,B 0,C 180,E1 -23637.672,E2 -23637.672} C_VEL
LIN {X 0,Y 155.615,Z 608.858,A -85,B 0,C 180,E1 -23643.155,E2 -23643.155} C_VEL
LIN {X 0,Y 155.001,Z 608.737,A -85,B 0,C 180,E1 -23645.919,E2 -23645.919} C_VEL
LIN {X 0,Y 154.412,Z 607.414,A -85,B 0,C 180,E1 -23651.424,E2 -23651.424} C_VEL
LIN {X 0,Y 154.439,Z 606.201,A -85,B 0,C 180,E1 -23654.157,E2 -23654.157} C_VEL
LIN {X 0,Y 155.066,Z 602.657,A -85,B 0,C 180,E1 -23659.558,E2 -23659.558} C_VEL
LIN {X 0,Y 156.118,Z 598.694,A -85,B 0,C 180,E1 -23663.857,E2 -23663.857} C_VEL
LIN {X 0,Y 157.889,Z 592.707,A -85,B 0,C 180,E1 -23668.727,E2 -23668.727} C_VEL
LIN {X 0,Y 160.31,Z 585.643,A -85,B 0,C 180,E1 -23673.144,E2 -23673.144} C_VEL
LIN {X 0,Y 163.481,Z 576.886,A -85,B 0,C 180,E1 -23677.412,E2 -23677.412} C_VEL
LIN {X 0,Y 166.706,Z 567.743,A -85,B 0,C 180,E1 -23680.938,E2 -23680.938} C_VEL
LIN {X 0,Y 170.48,Z 556.661,A -85,B 0,C 180,E1 -23684.323,E2 -23684.323} C_VEL
LIN {X 0,Y 174.054,Z 545.338,A -85,B 0,C 180,E1 -23687.024,E2 -23687.024} C_VEL
LIN {X 0,Y 177.613,Z 532.774,A -85,B 0,C 180,E1 -23689.355,E2 -23689.355} C_VEL
LIN {X 0,Y 180.459,Z 520.794,A -85,B 0,C 180,E1 -23691.102,E2 -23691.102} C_VEL
LIN {X 0,Y 182.995,Z 507.481,A -85,B 0,C 180,E1 -23692.587,E2 -23692.587} C_VEL
LIN {X 0,Y 185.043,Z 493.202,A -85,B 0,C 180,E1 -23693.727,E2 -23693.727} C_VEL
LIN {X 0,Y 186.352,Z 479.506,A -85,B 0,C 180,E1 -23694.438,E2 -23694.438} C_VEL
LIN {X 0,Y 190.32,Z 416.188,A -85,B 0,C 180,E1 -23696.596,E2 -23696.596} C_VEL
LIN {X 0,Y 184.958,Z 404.526,A -85,B 0,C 180,E1 -23698.499,E2 -23698.499} C_VEL
LIN {X 0,Y 178.391,Z 392.102,A -85,B 0,C 180,E1 -23700.966,E2 -23700.966} C_VEL
LIN {X 0,Y 171.513,Z 380.706,A -85,B 0,C 180,E1 -23703.743,E2 -23703.743} C_VEL
LIN {X 0,Y 166.038,Z 372.612,A -85,B 0,C 180,E1 -23706.15,E2 -23706.15} C_VEL
LIN {X 0,Y 163.557,Z 369.022,A -85,B 0,C 180,E1 -23707.327,E2 -23707.327} C_VEL
LIN {X 0,Y 161.167,Z 365.821,A -85,B 0,C 180,E1 -23708.504,E2 -23708.504} C_VEL
LIN {X 0,Y 160.473,Z 364.616,A -85,B 0,C 180,E1 -23708.877,E2 -23708.877} C_VEL
LIN {X 0,Y 158.255,Z 362.404,A -85,B 0,C 180,E1 -23709.993,E2 -23709.993} C_VEL
LIN {X 0,Y 157.315,Z 360.096,A -85,B 0,C 180,E1 -23710.584,E2 -23710.584} C_VEL
LIN {X 0,Y 157.209,Z 359.526,A -85,B 0,C 180,E1 -23710.769,E2 -23710.769} C_VEL
LIN {X 0,Y 157.179,Z 359.498,A -85,B 0,C 180,E1 -23715.68,E2 -23715.68} C_VEL
LIN {X 0,Y 157.199,Z 359.502,A -85,B 0,C 180,E1 -23721.252,E2 -23721.252} C_VEL
LIN {X 0,Y 157.276,Z 359.471,A -85,B 0,C 180,E1 -23724.486,E2 -23724.486} C_VEL
LIN {X 0,Y 157.286,Z 359.512,A -85,B 0,C 180,E1 -23728.104,E2 -23728.104} C_VEL
LIN {X 0,Y 157.313,Z 359.506,A -85,B 0,C 180,E1 -23733.466,E2 -23733.466} C_VEL
LIN {X 0,Y 157.363,Z 359.501,A -85,B 0,C 180,E1 -23739.704,E2 -23739.704} C_VEL
LIN {X 0,Y 157.409,Z 359.473,A -85,B 0,C 180,E1 -23744.462,E2 -23744.462} C_VEL
LIN {X 0,Y 157.69,Z 359.426,A -85,B 0,C 180,E1 -23749.732,E2 -23749.732} C_VEL
LIN {X 0,Y 157.763,Z 359.452,A -85,B 0,C 180,E1 -23752.321,E2 -23752.321} C_VEL
LIN {X 0,Y 158.251,Z 359.345,A -85,B 0,C 180,E1 -23760.001,E2 -23760.001} C_VEL
LIN {X 0,Y 157.767,Z 359.448,A -85,B 0,C 180,E1 -23767.681,E2 -23767.681} C_VEL
LIN {X 0,Y 157.643,Z 359.474,A -85,B 0,C 180,E1 -23771.236,E2 -23771.236} C_VEL
LIN {X 0,Y 157.448,Z 359.494,A -85,B 0,C 180,E1 -23775.536,E2 -23775.536} C_VEL
LIN {X 0,Y 157.376,Z 359.497,A -85,B 0,C 180,E1 -23780.933,E2 -23780.933} C_VEL
LIN {X 0,Y 157.317,Z 359.507,A -85,B 0,C 180,E1 -23786.681,E2 -23786.681} C_VEL
LIN {X 0,Y 157.35,Z 359.502,A -85,B 0,C 180,E1 -23790.815,E2 -23790.815} C_VEL
LIN {X 0,Y 158.293,Z 362.292,A -85,B 0,C 180,E1 -23791.478,E2 -23791.478} C_VEL
LIN {X 0,Y 160.348,Z 364.468,A -85,B 0,C 180,E1 -23792.522,E2 -23792.522} C_VEL
LIN {X 0,Y 161.087,Z 365.625,A -85,B 0,C 180,E1 -23792.91,E2 -23792.91} C_VEL
LIN {X 0,Y 163.312,Z 368.73,A -85,B 0,C 180,E1 -23794.018,E2 -23794.018} C_VEL
LIN {X 0,Y 167.643,Z 374.956,A -85,B 0,C 180,E1 -23796.043,E2 -23796.043} C_VEL
LIN {X 0,Y 170.834,Z 379.921,A -85,B 0,C 180,E1 -23797.452,E2 -23797.452} C_VEL
LIN {X 0,Y 176.06,Z 390.059,A -85,B 0,C 180,E1 -23799.695,E2 -23799.695} C_VEL
LIN {X 0,Y 181.786,Z 402.857,A -85,B 0,C 180,E1 -23802.04,E2 -23802.04} C_VEL
LIN {X 0,Y 187.354,Z 417.504,A -85,B 0,C 180,E1 -23804.223,E2 -23804.223} C_VEL
LIN {X 0,Y 189.497,Z 424.522,A -85,B 0,C 180,E1 -23805.079,E2 -23805.079} C_VEL
LIN {X 0,Y 189.697,Z 429.407,A -85,B 0,C 180,E1 -23805.361,E2 -23805.361} C_VEL
LIN {X 0,Y 185.597,Z 495.447,A -85,B 0,C 180,E1 -23807.674,E2 -23807.674} C_VEL
LIN {X 0,Y 183.945,Z 509.29,A -85,B 0,C 180,E1 -23808.495,E2 -23808.495} C_VEL
LIN {X 0,Y 181.531,Z 523.52,A -85,B 0,C 180,E1 -23809.753,E2 -23809.753} C_VEL
LIN {X 0,Y 178.527,Z 536.665,A -85,B 0,C 180,E1 -23811.32,E2 -23811.32} C_VEL
LIN {X 0,Y 175.576,Z 547.992,A -85,B 0,C 180,E1 -23813.098,E2 -23813.098} C_VEL
LIN {X 0,Y 173.043,Z 556.951,A -85,B 0,C 180,E1 -23814.832,E2 -23814.832} C_VEL
LIN {X 0,Y 171.756,Z 560.755,A -85,B 0,C 180,E1 -23815.665,E2 -23815.665} C_VEL
LIN {X 0,Y 169.506,Z 565.395,A -85,B 0,C 180,E1 -23816.646,E2 -23816.646} C_VEL
LIN {X 0,Y 164.394,Z 572.592,A -85,B 0,C 180,E1 -23818.208,E2 -23818.208} C_VEL
LIN {X 0,Y 159.366,Z 579.322,A -85,B 0,C 180,E1 -23820.058,E2 -23820.058} C_VEL
LIN {X 0,Y 157.294,Z 583.224,A -85,B 0,C 180,E1 -23821.473,E2 -23821.473} C_VEL
LIN {X 0,Y 154.301,Z 591.423,A -85,B 0,C 180,E1 -23825.08,E2 -23825.08} C_VEL
LIN {X 0,Y 151.791,Z 598.556,A -85,B 0,C 180,E1 -23828.969,E2 -23828.969} C_VEL
LIN {X 0,Y 149.607,Z 605.306,A -85,B 0,C 180,E1 -23833.626,E2 -23833.626} C_VEL
LIN {X 0,Y 148.213,Z 611.269,A -85,B 0,C 180,E1 -23839.064,E2 -23839.064} C_VEL
LIN {X 0,Y 147.887,Z 613.626,A -85,B 0,C 180,E1 -23841.801,E2 -23841.801} C_VEL
LIN {X 0,Y 147.744,Z 615.59,A -85,B 0,C 180,E1 -23844.538,E2 -23844.538} C_VEL
LIN {X 0,Y 147.758,Z 617.178,A -85,B 0,C 180,E1 -23847.271,E2 -23847.271} C_VEL
LIN {X 0,Y 147.893,Z 618.403,A -85,B 0,C 180,E1 -23849.998,E2 -23849.998} C_VEL
LIN {X 0,Y 147.757,Z 619.255,A -85,B 0,C 180,E1 -23852.724,E2 -23852.724} C_VEL
LIN {X 0,Y 147.837,Z 619.948,A -85,B 0,C 180,E1 -23858.197,E2 -23858.197} C_VEL
LIN {X 0,Y 148.889,Z 619.34,A -85,B 0,C 180,E1 -23863.649,E2 -23863.649} C_VEL
LIN {X 0,Y 151.16,Z 617.443,A -85,B 0,C 180,E1 -23868.991,E2 -23868.991} C_VEL
LIN {X 0,Y 154.602,Z 614.221,A -85,B 0,C 180,E1 -23874.147,E2 -23874.147} C_VEL
LIN {X 0,Y 159.281,Z 609.575,A -85,B 0,C 180,E1 -23879.033,E2 -23879.033} C_VEL
LIN {X 0,Y 165.125,Z 603.336,A -85,B 0,C 180,E1 -23883.591,E2 -23883.591} C_VEL
LIN {X 0,Y 171.095,Z 596.461,A -85,B 0,C 180,E1 -23887.289,E2 -23887.289} C_VEL
LIN {X 0,Y 177.879,Z 587.976,A -85,B 0,C 180,E1 -23890.683,E2 -23890.683} C_VEL
LIN {X 0,Y 184.066,Z 579.18,A -85,B 0,C 180,E1 -23893.412,E2 -23893.412} C_VEL
LIN {X 0,Y 190.757,Z 568.564,A -85,B 0,C 180,E1 -23895.922,E2 -23895.922} C_VEL
LIN {X 0,Y 196.625,Z 557.876,A -85,B 0,C 180,E1 -23897.871,E2 -23897.871} C_VEL
LIN {X 0,Y 202.099,Z 546.247,A -85,B 0,C 180,E1 -23899.523,E2 -23899.523} C_VEL
LIN {X 0,Y 207.228,Z 533.445,A -85,B 0,C 180,E1 -23900.873,E2 -23900.873} C_VEL
LIN {X 0,Y 211.384,Z 520.221,A -85,B 0,C 180,E1 -23901.954,E2 -23901.954} C_VEL
LIN {X 0,Y 214.925,Z 505.623,A -85,B 0,C 180,E1 -23902.756,E2 -23902.756} C_VEL
LIN {X 0,Y 217.096,Z 491.71,A -85,B 0,C 180,E1 -23903.307,E2 -23903.307} C_VEL
LIN {X 0,Y 220.551,Z 452.956,A -85,B 0,C 180,E1 -23904.382,E2 -23904.382} C_VEL
LIN {X 0,Y 216.957,Z 443.926,A -85,B 0,C 180,E1 -23906.871,E2 -23906.871} C_VEL
LIN {X 0,Y 213.289,Z 435.687,A -85,B 0,C 180,E1 -23909.691,E2 -23909.691} C_VEL
LIN {X 0,Y 210.287,Z 429.295,A -85,B 0,C 180,E1 -23912.397,E2 -23912.397} C_VEL
LIN {X 0,Y 207.901,Z 424.492,A -85,B 0,C 180,E1 -23914.869,E2 -23914.869} C_VEL
LIN {X 0,Y 205.331,Z 419.767,A -85,B 0,C 180,E1 -23918.007,E2 -23918.007} C_VEL
LIN {X 0,Y 202.762,Z 414.809,A -85,B 0,C 180,E1 -23922.368,E2 -23922.368} C_VEL
LIN {X 0,Y 200.562,Z 411.782,A -85,B 0,C 180,E1 -23930.597,E2 -23930.597} C_VEL
LIN {X 0,Y 200.577,Z 411.791,A -85,B 0,C 180,E1 -23932.282,E2 -23932.282} C_VEL
LIN {X 0,Y 202.704,Z 414.418,A -85,B 0,C 180,E1 -23939.999,E2 -23939.999} C_VEL
LIN {X 0,Y 205.353,Z 418.801,A -85,B 0,C 180,E1 -23944.445,E2 -23944.445} C_VEL
LIN {X 0,Y 206.533,Z 420.852,A -85,B 0,C 180,E1 -23945.965,E2 -23945.965} C_VEL
LIN {X 0,Y 208.859,Z 424.334,A -85,B 0,C 180,E1 -23948.499,E2 -23948.499} C_VEL
LIN {X 0,Y 212.29,Z 430.02,A -85,B 0,C 180,E1 -23951.683,E2 -23951.683} C_VEL
LIN {X 0,Y 216.033,Z 436.497,A -85,B 0,C 180,E1 -23954.6,E2 -23954.6} C_VEL
LIN {X 0,Y 220.227,Z 444.296,A -85,B 0,C 180,E1 -23957.417,E2 -23957.417} C_VEL
LIN {X 0,Y 221.038,Z 445.892,A -85,B 0,C 180,E1 -23957.926,E2 -23957.926} C_VEL
LIN {X 0,Y 217.463,Z 485.893,A -85,B 0,C 180,E1 -23959.082,E2 -23959.082} C_VEL
LIN {X 0,Y 215.266,Z 499.24,A -85,B 0,C 180,E1 -23959.669,E2 -23959.669} C_VEL
LIN {X 0,Y 212.037,Z 512.939,A -85,B 0,C 180,E1 -23960.559,E2 -23960.559} C_VEL
LIN {X 0,Y 208.056,Z 525.838,A -85,B 0,C 180,E1 -23961.705,E2 -23961.705} C_VEL
LIN {X 0,Y 203.46,Z 537.909,A -85,B 0,C 180,E1 -23963.125,E2 -23963.125} C_VEL
LIN {X 0,Y 197.935,Z 549.785,A -85,B 0,C 180,E1 -23964.891,E2 -23964.891} C_VEL
LIN {X 0,Y 192.172,Z 560.442,A -85,B 0,C 180,E1 -23966.952,E2 -23966.952} C_VEL
LIN {X 0,Y 185.703,Z 570.734,A -85,B 0,C 180,E1 -23969.495,E2 -23969.495} C_VEL
LIN {X 0,Y 179.107,Z 579.964,A -85,B 0,C 180,E1 -23972.478,E2 -23972.478} C_VEL
LIN {X 0,Y 172.06,Z 588.639,A -85,B 0,C 180,E1 -23976.228,E2 -23976.228} C_VEL
LIN {X 0,Y 165.779,Z 595.473,A -85,B 0,C 180,E1 -23980.267,E2 -23980.267} C_VEL
LIN {X 0,Y 160.61,Z 600.6,A -85,B 0,C 180,E1 -23984.436,E2 -23984.436} C_VEL
LIN {X 0,Y 157.151,Z 603.738,A -85,B 0,C 180,E1 -23987.873,E2 -23987.873} C_VEL
LIN {X 0,Y 154.868,Z 605.612,A -85,B 0,C 180,E1 -23990.559,E2 -23990.559} C_VEL
LIN {X 0,Y 151.258,Z 608.117,A -85,B 0,C 180,E1 -23996.116,E2 -23996.116} C_VEL
LIN {X 0,Y 148.881,Z 609.109,A -85,B 0,C 180,E1 -24001.835,E2 -24001.835} C_VEL
LIN {X 0,Y 148.139,Z 609.053,A -85,B 0,C 180,E1 -24004.727,E2 -24004.727} C_VEL
LIN {X 0,Y 147.325,Z 607.863,A -85,B 0,C 180,E1 -24010.495,E2 -24010.495} C_VEL
LIN {X 0,Y 147.316,Z 606.727,A -85,B 0,C 180,E1 -24013.37,E2 -24013.37} C_VEL
LIN {X 0,Y 147.853,Z 603.36,A -85,B 0,C 180,E1 -24019.042,E2 -24019.042} C_VEL
LIN {X 0,Y 148.715,Z 600.072,A -85,B 0,C 180,E1 -24022.933,E2 -24022.933} C_VEL
LIN {X 0,Y 150.147,Z 595.352,A -85,B 0,C 180,E1 -24027.32,E2 -24027.32} C_VEL
LIN {X 0,Y 152.321,Z 588.899,A -85,B 0,C 180,E1 -24031.985,E2 -24031.985} C_VEL
LIN {X 0,Y 155.331,Z 581.012,A -85,B 0,C 180,E1 -24036.414,E2 -24036.414} C_VEL
LIN {X 0,Y 158.508,Z 572.462,A -85,B 0,C 180,E1 -24040.218,E2 -24040.218} C_VEL
LIN {X 0,Y 162.199,Z 562.345,A -85,B 0,C 180,E1 -24043.789,E2 -24043.789} C_VEL
LIN {X 0,Y 166.183,Z 551.007,A -85,B 0,C 180,E1 -24046.905,E2 -24046.905} C_VEL
LIN {X 0,Y 169.649,Z 539.738,A -85,B 0,C 180,E1 -24049.357,E2 -24049.357} C_VEL
LIN {X 0,Y 172.996,Z 527.433,A -85,B 0,C 180,E1 -24051.448,E2 -24051.448} C_VEL
LIN {X 0,Y 175.854,Z 514.763,A -85,B 0,C 180,E1 -24053.112,E2 -24053.112} C_VEL
LIN {X 0,Y 178.311,Z 500.309,A -85,B 0,C 180,E1 -24054.527,E2 -24054.527} C_VEL
LIN {X 0,Y 180.144,Z 485.809,A -85,B 0,C 180,E1 -24055.466,E2 -24055.466} C_VEL
LIN {X 0,Y 182.152,Z 457.345,A -85,B 0,C 180,E1 -24056.527,E2 -24056.527} C_VEL
LIN {X 0,Y 184.582,Z 418.003,A -85,B 0,C 180,E1 -24057.909,E2 -24057.909} C_VEL
LIN {X 0,Y 177.361,Z 402.81,A -85,B 0,C 180,E1 -24060.678,E2 -24060.678} C_VEL
LIN {X 0,Y 170.949,Z 391.344,A -85,B 0,C 180,E1 -24063.296,E2 -24063.296} C_VEL
LIN {X 0,Y 164.812,Z 381.536,A -85,B 0,C 180,E1 -24066.029,E2 -24066.029} C_VEL
LIN {X 0,Y 160.003,Z 374.485,A -85,B 0,C 180,E1 -24068.385,E2 -24068.385} C_VEL
LIN {X 0,Y 157.446,Z 370.792,A -85,B 0,C 180,E1 -24069.742,E2 -24069.742} C_VEL
LIN {X 0,Y 154.551,Z 367.275,A -85,B 0,C 180,E1 -24071.328,E2 -24071.328} C_VEL
LIN {X 0,Y 153.565,Z 365.618,A -85,B 0,C 180,E1 -24071.927,E2 -24071.927} C_VEL
LIN {X 0,Y 151.282,Z 363.489,A -85,B 0,C 180,E1 -24073.24,E2 -24073.24} C_VEL
LIN {X 0,Y 150.269,Z 361.14,A -85,B 0,C 180,E1 -24073.965,E2 -24073.965} C_VEL
LIN {X 0,Y 150.124,Z 360.371,A -85,B 0,C 180,E1 -24074.112,E2 -24074.112} C_VEL
LIN {X 0,Y 150.139,Z 360.406,A -85,B 0,C 180,E1 -24079.056,E2 -24079.056} C_VEL
LIN {X 0,Y 150.178,Z 360.357,A -85,B 0,C 180,E1 -24082.712,E2 -24082.712} C_VEL
LIN {X 0,Y 150.211,Z 360.382,A -85,B 0,C 180,E1 -24087.374,E2 -24087.374} C_VEL
LIN {X 0,Y 150.231,Z 360.384,A -85,B 0,C 180,E1 -24092.732,E2 -24092.732} C_VEL
LIN {X 0,Y 150.287,Z 360.379,A -85,B 0,C 180,E1 -24099.279,E2 -24099.279} C_VEL
LIN {X 0,Y 150.315,Z 360.367,A -85,B 0,C 180,E1 -24103.709,E2 -24103.709} C_VEL
LIN {X 0,Y 150.61,Z 360.3,A -85,B 0,C 180,E1 -24109.243,E2 -24109.243} C_VEL
LIN {X 0,Y 150.702,Z 360.328,A -85,B 0,C 180,E1 -24111.959,E2 -24111.959} C_VEL
LIN {X 0,Y 151.21,Z 360.22,A -85,B 0,C 180,E1 -24120.001,E2 -24120.001} C_VEL
LIN {X 0,Y 150.689,Z 360.328,A -85,B 0,C 180,E1 -24128.044,E2 -24128.044} C_VEL
LIN {X 0,Y 150.583,Z 360.354,A -85,B 0,C 180,E1 -24131.437,E2 -24131.437} C_VEL
LIN {X 0,Y 150.36,Z 360.381,A -85,B 0,C 180,E1 -24136.288,E2 -24136.288} C_VEL
LIN {X 0,Y 150.357,Z 360.369,A -85,B 0,C 180,E1 -24140.792,E2 -24140.792} C_VEL
LIN {X 0,Y 150.245,Z 360.392,A -85,B 0,C 180,E1 -24147.407,E2 -24147.407} C_VEL
LIN {X 0,Y 151.096,Z 363.046,A -85,B 0,C 180,E1 -24148.097,E2 -24148.097} C_VEL
LIN {X 0,Y 153.13,Z 365.275,A -85,B 0,C 180,E1 -24149.302,E2 -24149.302} C_VEL
LIN {X 0,Y 154.094,Z 366.059,A -85,B 0,C 180,E1 -24149.83,E2 -24149.83} C_VEL
LIN {X 0,Y 156.043,Z 369.254,A -85,B 0,C 180,E1 -24150.978,E2 -24150.978} C_VEL
LIN {X 0,Y 157.607,Z 371.044,A -85,B 0,C 180,E1 -24151.811,E2 -24151.811} C_VEL
LIN {X 0,Y 160.139,Z 374.613,A -85,B 0,C 180,E1 -24153.142,E2 -24153.142} C_VEL
LIN {X 0,Y 166.059,Z 383.452,A -85,B 0,C 180,E1 -24156.009,E2 -24156.009} C_VEL
LIN {X 0,Y 171.213,Z 393.487,A -85,B 0,C 180,E1 -24158.379,E2 -24158.379} C_VEL
LIN {X 0,Y 176.958,Z 406.58,A -85,B 0,C 180,E1 -24160.881,E2 -24160.881} C_VEL
LIN {X 0,Y 182.288,Z 420.929,A -85,B 0,C 180,E1 -24163.117,E2 -24163.117} C_VEL
LIN {X 0,Y 183.98,Z 426.36,A -85,B 0,C 180,E1 -24163.829,E2 -24163.829} C_VEL
LIN {X 0,Y 184.072,Z 430.04,A -85,B 0,C 180,E1 -24164.038,E2 -24164.038} C_VEL
LIN {X 0,Y 179.854,Z 495.325,A -85,B 0,C 180,E1 -24166.372,E2 -24166.372} C_VEL
LIN {X 0,Y 178.022,Z 509.89,A -85,B 0,C 180,E1 -24167.269,E2 -24167.269} C_VEL
LIN {X 0,Y 175.38,Z 524.457,A -85,B 0,C 180,E1 -24168.606,E2 -24168.606} C_VEL
LIN {X 0,Y 172.08,Z 538.246,A -85,B 0,C 180,E1 -24170.344,E2 -24170.344} C_VEL
LIN {X 0,Y 168.439,Z 551.165,A -85,B 0,C 180,E1 -24172.525,E2 -24172.525} C_VEL
LIN {X 0,Y 165.368,Z 560.845,A -85,B 0,C 180,E1 -24174.614,E2 -24174.614} C_VEL
LIN {X 0,Y 162.024,Z 570.51,A -85,B 0,C 180,E1 -24177.164,E2 -24177.164} C_VEL
LIN {X 0,Y 158.019,Z 581.241,A -85,B 0,C 180,E1 -24180.707,E2 -24180.707} C_VEL
LIN {X 0,Y 157.294,Z 583.224,A -85,B 0,C 180,E1 -24181.473,E2 -24181.473} C_VEL
LIN {X 0,Y 155.246,Z 587.034,A -85,B 0,C 180,E1 -24182.971,E2 -24182.971} C_VEL
LIN {X 0,Y 150.353,Z 592.733,A -85,B 0,C 180,E1 -24185.386,E2 -24185.386} C_VEL
LIN {X 0,Y 145.649,Z 597.958,A -85,B 0,C 180,E1 -24188.096,E2 -24188.096} C_VEL
LIN {X 0,Y 143.961,Z 600.876,A -85,B 0,C 180,E1 -24190.017,E2 -24190.017} C_VEL
LIN {X 0,Y 142.234,Z 606.284,A -85,B 0,C 180,E1 -24194.228,E2 -24194.228} C_VEL
LIN {X 0,Y 140.988,Z 611.956,A -85,B 0,C 180,E1 -24199.95,E2 -24199.95} C_VEL
LIN {X 0,Y 140.677,Z 615.105,A -85,B 0,C 180,E1 -24204.263,E2 -24204.263} C_VEL
LIN {X 0,Y 140.819,Z 617.999,A -85,B 0,C 180,E1 -24209.997,E2 -24209.997} C_VEL
LIN {X 0,Y 140.657,Z 618.888,A -85,B 0,C 180,E1 -24212.861,E2 -24212.861} C_VEL
LIN {X 0,Y 140.788,Z 619.658,A -85,B 0,C 180,E1 -24218.61,E2 -24218.61} C_VEL
LIN {X 0,Y 141.956,Z 619.126,A -85,B 0,C 180,E1 -24224.329,E2 -24224.329} C_VEL
LIN {X 0,Y 144.429,Z 617.308,A -85,B 0,C 180,E1 -24229.912,E2 -24229.912} C_VEL
LIN {X 0,Y 148.091,Z 614.166,A -85,B 0,C 180,E1 -24235.282,E2 -24235.282} C_VEL
LIN {X 0,Y 153.085,Z 609.632,A -85,B 0,C 180,E1 -24240.328,E2 -24240.328} C_VEL
LIN {X 0,Y 159.264,Z 603.54,A -85,B 0,C 180,E1 -24245.003,E2 -24245.003} C_VEL
LIN {X 0,Y 165.506,Z 596.776,A -85,B 0,C 180,E1 -24248.777,E2 -24248.777} C_VEL
LIN {X 0,Y 172.58,Z 588.414,A -85,B 0,C 180,E1 -24252.213,E2 -24252.213} C_VEL
LIN {X 0,Y 178.992,Z 579.76,A -85,B 0,C 180,E1 -24254.968,E2 -24254.968} C_VEL
LIN {X 0,Y 185.911,Z 569.313,A -85,B 0,C 180,E1 -24257.487,E2 -24257.487} C_VEL
LIN {X 0,Y 191.975,Z 558.827,A -85,B 0,C 180,E1 -24259.429,E2 -24259.429} C_VEL
LIN {X 0,Y 197.614,Z 547.455,A -85,B 0,C 180,E1 -24261.072,E2 -24261.072} C_VEL
LIN {X 0,Y 202.881,Z 535.002,A -85,B 0,C 180,E1 -24262.408,E2 -24262.408} C_VEL
LIN {X 0,Y 207.475,Z 521.172,A -85,B 0,C 180,E1 -24263.559,E2 -24263.559} C_VEL
LIN {X 0,Y 211.103,Z 507.187,A -85,B 0,C 180,E1 -24264.342,E2 -24264.342} C_VEL
LIN {X 0,Y 213.567,Z 492.716,A -85,B 0,C 180,E1 -24264.934,E2 -24264.934} C_VEL
LIN {X 0,Y 216.94,Z 456.029,A -85,B 0,C 180,E1 -24265.969,E2 -24265.969} C_VEL
LIN {X 0,Y 213.83,Z 447.993,A -85,B 0,C 180,E1 -24268.316,E2 -24268.316} C_VEL
LIN {X 0,Y 210.381,Z 439.702,A -85,B 0,C 180,E1 -24271.296,E2 -24271.296} C_VEL
LIN {X 0,Y 207.801,Z 434.26,A -85,B 0,C 180,E1 -24273.841,E2 -24273.841} C_VEL
LIN {X 0,Y 206.22,Z 430.834,A -85,B 0,C 180,E1 -24275.634,E2 -24275.634} C_VEL
LIN {X 0,Y 203.86,Z 426.258,A -85,B 0,C 180,E1 -24278.719,E2 -24278.719} C_VEL
LIN {X 0,Y 201.627,Z 421.727,A -85,B 0,C 180,E1 -24282.813,E2 -24282.813} C_VEL
LIN {X 0,Y 199.651,Z 418.776,A -85,B 0,C 180,E1 -24291.23,E2 -24291.23} C_VEL
LIN {X 0,Y 199.782,Z 419.224,A -85,B 0,C 180,E1 -24293.519,E2 -24293.519} C_VEL
LIN {X 0,Y 201.706,Z 421.4,A -85,B 0,C 180,E1 -24299.812,E2 -24299.812} C_VEL
LIN {X 0,Y 203.919,Z 425.446,A -85,B 0,C 180,E1 -24303.796,E2 -24303.796} C_VEL
LIN {X 0,Y 204.775,Z 426.866,A -85,B 0,C 180,E1 -24304.965,E2 -24304.965} C_VEL
LIN {X 0,Y 207.31,Z 430.998,A -85,B 0,C 180,E1 -24307.932,E2 -24307.932} C_VEL
LIN {X 0,Y 209.785,Z 435.301,A -85,B 0,C 180,E1 -24310.394,E2 -24310.394} C_VEL
LIN {X 0,Y 213.047,Z 441.066,A -85,B 0,C 180,E1 -24313.188,E2 -24313.188} C_VEL
LIN {X 0,Y 217.251,Z 449.142,A -85,B 0,C 180,E1 -24316.246,E2 -24316.246} C_VEL
LIN {X 0,Y 217.483,Z 449.624,A -85,B 0,C 180,E1 -24316.404,E2 -24316.404} C_VEL
LIN {X 0,Y 214.079,Z 486.004,A -85,B 0,C 180,E1 -24317.43,E2 -24317.43} C_VEL
LIN {X 0,Y 211.764,Z 499.578,A -85,B 0,C 180,E1 -24318.01,E2 -24318.01} C_VEL
LIN {X 0,Y 208.441,Z 513.264,A -85,B 0,C 180,E1 -24318.889,E2 -24318.889} C_VEL
LIN {X 0,Y 204.267,Z 526.349,A -85,B 0,C 180,E1 -24320.043,E2 -24320.043} C_VEL
LIN {X 0,Y 199.253,Z 538.97,A -85,B 0,C 180,E1 -24321.526,E2 -24321.526} C_VEL
LIN {X 0,Y 193.176,Z 551.447,A -85,B 0,C 180,E1 -24323.412,E2 -24323.412} C_VEL
LIN {X 0,Y 186.962,Z 562.285,A -85,B 0,C 180,E1 -24325.561,E2 -24325.561} C_VEL
LIN {X 0,Y 180.632,Z 571.807,A -85,B 0,C 180,E1 -24327.981,E2 -24327.981} C_VEL
LIN {X 0,Y 173.999,Z 580.603,A -85,B 0,C 180,E1 -24330.878,E2 -24330.878} C_VEL
LIN {X 0,Y 167.632,Z 588.093,A -85,B 0,C 180,E1 -24334.109,E2 -24334.109} C_VEL
LIN {X 0,Y 160.941,Z 595.118,A -85,B 0,C 180,E1 -24338.188,E2 -24338.188} C_VEL
LIN {X 0,Y 154.649,Z 600.947,A -85,B 0,C 180,E1 -24342.973,E2 -24342.973} C_VEL
LIN {X 0,Y 151.528,Z 603.586,A -85,B 0,C 180,E1 -24345.92,E2 -24345.92} C_VEL
LIN {X 0,Y 148.563,Z 605.869,A -85,B 0,C 180,E1 -24349.191,E2 -24349.191} C_VEL
LIN {X 0,Y 144.956,Z 608.235,A -85,B 0,C 180,E1 -24354.426,E2 -24354.426} C_VEL
LIN {X 0,Y 142.2,Z 609.362,A -85,B 0,C 180,E1 -24360.384,E2 -24360.384} C_VEL
LIN {X 0,Y 140.676,Z 609.019,A -85,B 0,C 180,E1 -24366.446,E2 -24366.446} C_VEL
LIN {X 0,Y 140.211,Z 607.235,A -85,B 0,C 180,E1 -24372.5,E2 -24372.5} C_VEL
LIN {X 0,Y 140.636,Z 604.013,A -85,B 0,C 180,E1 -24378.472,E2 -24378.472} C_VEL
LIN {X 0,Y 141.614,Z 600.465,A -85,B 0,C 180,E1 -24382.995,E2 -24382.995} C_VEL
LIN {X 0,Y 143.486,Z 594.611,A -85,B 0,C 180,E1 -24388.599,E2 -24388.599} C_VEL
LIN {X 0,Y 145.925,Z 587.909,A -85,B 0,C 180,E1 -24393.454,E2 -24393.454} C_VEL
LIN {X 0,Y 149.264,Z 579.555,A -85,B 0,C 180,E1 -24398.123,E2 -24398.123} C_VEL
LIN {X 0,Y 152.693,Z 570.831,A -85,B 0,C 180,E1 -24401.956,E2 -24401.956} C_VEL
LIN {X 0,Y 156.665,Z 560.257,A -85,B 0,C 180,E1 -24405.617,E2 -24405.617} C_VEL
LIN {X 0,Y 160.858,Z 548.396,A -85,B 0,C 180,E1 -24408.799,E2 -24408.799} C_VEL
LIN {X 0,Y 164.648,Z 536.48,A -85,B 0,C 180,E1 -24411.276,E2 -24411.276} C_VEL
LIN {X 0,Y 167.853,Z 524.6,A -85,B 0,C 180,E1 -24413.212,E2 -24413.212} C_VEL
LIN {X 0,Y 170.748,Z 511.57,A -85,B 0,C 180,E1 -24414.843,E2 -24414.843} C_VEL
LIN {X 0,Y 173.044,Z 497.52,A -85,B 0,C 180,E1 -24416.154,E2 -24416.154} C_VEL
LIN {X 0,Y 174.701,Z 483.937,A -85,B 0,C 180,E1 -24416.973,E2 -24416.973} C_VEL
LIN {X 0,Y 179.085,Z 420.393,A -85,B 0,C 180,E1 -24419.237,E2 -24419.237} C_VEL
LIN {X 0,Y 172.131,Z 405.766,A -85,B 0,C 180,E1 -24422.079,E2 -24422.079} C_VEL
LIN {X 0,Y 165.501,Z 393.821,A -85,B 0,C 180,E1 -24424.996,E2 -24424.996} C_VEL
LIN {X 0,Y 159.142,Z 383.731,A -85,B 0,C 180,E1 -24428.098,E2 -24428.098} C_VEL
LIN {X 0,Y 155.742,Z 378.948,A -85,B 0,C 180,E1 -24429.904,E2 -24429.904} C_VEL
LIN {X 0,Y 153.426,Z 375.631,A -85,B 0,C 180,E1 -24431.226,E2 -24431.226} C_VEL
LIN {X 0,Y 150.343,Z 371.466,A -85,B 0,C 180,E1 -24433.081,E2 -24433.081} C_VEL
LIN {X 0,Y 147.873,Z 368.554,A -85,B 0,C 180,E1 -24434.651,E2 -24434.651} C_VEL
LIN {X 0,Y 146.898,Z 366.696,A -85,B 0,C 180,E1 -24435.36,E2 -24435.36} C_VEL
LIN {X 0,Y 144.492,Z 364.774,A -85,B 0,C 180,E1 -24436.958,E2 -24436.958} C_VEL
LIN {X 0,Y 143.274,Z 362.351,A -85,B 0,C 180,E1 -24437.954,E2 -24437.954} C_VEL
LIN {X 0,Y 143.072,Z 361.283,A -85,B 0,C 180,E1 -24438.211,E2 -24438.211} C_VEL
LIN {X 0,Y 143.084,Z 361.235,A -85,B 0,C 180,E1 -24443.886,E2 -24443.886} C_VEL
LIN {X 0,Y 143.178,Z 361.254,A -85,B 0,C 180,E1 -24447.321,E2 -24447.321} C_VEL
LIN {X 0,Y 143.179,Z 361.262,A -85,B 0,C 180,E1 -24452.076,E2 -24452.076} C_VEL
LIN {X 0,Y 143.225,Z 361.256,A -85,B 0,C 180,E1 -24458.806,E2 -24458.806} C_VEL
LIN {X 0,Y 143.255,Z 361.256,A -85,B 0,C 180,E1 -24462.882,E2 -24462.882} C_VEL
LIN {X 0,Y 143.536,Z 361.174,A -85,B 0,C 180,E1 -24468.706,E2 -24468.706} C_VEL
LIN {X 0,Y 143.624,Z 361.202,A -85,B 0,C 180,E1 -24471.559,E2 -24471.559} C_VEL
LIN {X 0,Y 144.168,Z 361.095,A -85,B 0,C 180,E1 -24480.001,E2 -24480.001} C_VEL
LIN {X 0,Y 143.615,Z 361.208,A -85,B 0,C 180,E1 -24488.443,E2 -24488.443} C_VEL
LIN {X 0,Y 143.51,Z 361.233,A -85,B 0,C 180,E1 -24491.628,E2 -24491.628} C_VEL
LIN {X 0,Y 143.303,Z 361.259,A -85,B 0,C 180,E1 -24497.114,E2 -24497.114} C_VEL
LIN {X 0,Y 143.283,Z 361.253,A -85,B 0,C 180,E1 -24501.254,E2 -24501.254} C_VEL
LIN {X 0,Y 143.165,Z 361.269,A -85,B 0,C 180,E1 -24503.316,E2 -24503.316} C_VEL
LIN {X 0,Y 144.026,Z 363.868,A -85,B 0,C 180,E1 -24504.122,E2 -24504.122} C_VEL
LIN {X 0,Y 146.17,Z 366.227,A -85,B 0,C 180,E1 -24505.642,E2 -24505.642} C_VEL
LIN {X 0,Y 147.26,Z 367.091,A -85,B 0,C 180,E1 -24506.349,E2 -24506.349} C_VEL
LIN {X 0,Y 149.136,Z 370.201,A -85,B 0,C 180,E1 -24507.649,E2 -24507.649} C_VEL
LIN {X 0,Y 151.118,Z 372.287,A -85,B 0,C 180,E1 -24508.85,E2 -24508.85} C_VEL
LIN {X 0,Y 153.739,Z 375.891,A -85,B 0,C 180,E1 -24510.408,E2 -24510.408} C_VEL
LIN {X 0,Y 158.304,Z 382.586,A -85,B 0,C 180,E1 -24512.935,E2 -24512.935} C_VEL
LIN {X 0,Y 162.507,Z 389.086,A -85,B 0,C 180,E1 -24515.058,E2 -24515.058} C_VEL
LIN {X 0,Y 167.144,Z 398.552,A -85,B 0,C 180,E1 -24517.331,E2 -24517.331} C_VEL
LIN {X 0,Y 172.586,Z 411.323,A -85,B 0,C 180,E1 -24519.839,E2 -24519.839} C_VEL
LIN {X 0,Y 177.541,Z 425.191,A -85,B 0,C 180,E1 -24522.061,E2 -24522.061} C_VEL
LIN {X 0,Y 178.6,Z 428.768,A -85,B 0,C 180,E1 -24522.544,E2 -24522.544} C_VEL
LIN {X 0,Y 174.319,Z 493.94,A -85,B 0,C 180,E1 -24524.92,E2 -24524.92} C_VEL
LIN {X 0,Y 172.533,Z 508.167,A -85,B 0,C 180,E1 -24525.765,E2 -24525.765} C_VEL
LIN {X 0,Y 170.121,Z 522.009,A -85,B 0,C 180,E1 -24527.025,E2 -24527.025} C_VEL
LIN {X 0,Y 167.083,Z 534.458,A -85,B 0,C 180,E1 -24528.507,E2 -24528.507} C_VEL
LIN {X 0,Y 163.607,Z 546.895,A -85,B 0,C 180,E1 -24530.501,E2 -24530.501} C_VEL
LIN {X 0,Y 160.857,Z 555.766,A -85,B 0,C 180,E1 -24532.287,E2 -24532.287} C_VEL
LIN {X 0,Y 157.201,Z 566.2,A -85,B 0,C 180,E1 -24534.856,E2 -24534.856} C_VEL
LIN {X 0,Y 153.101,Z 576.804,A -85,B 0,C 180,E1 -24538.134,E2 -24538.134} C_VEL
LIN {X 0,Y 149.419,Z 586.39,A -85,B 0,C 180,E1 -24541.94,E2 -24541.94} C_VEL
LIN {X 0,Y 146.468,Z 594.004,A -85,B 0,C 180,E1 -24545.741,E2 -24545.741} C_VEL
LIN {X 0,Y 143.961,Z 600.876,A -85,B 0,C 180,E1 -24550.017,E2 -24550.017} C_VEL
LIN {X 0,Y 142.413,Z 603.651,A -85,B 0,C 180,E1 -24552.023,E2 -24552.023} C_VEL
LIN {X 0,Y 138.41,Z 607.635,A -85,B 0,C 180,E1 -24555.346,E2 -24555.346} C_VEL
LIN {X 0,Y 135.323,Z 610.398,A -85,B 0,C 180,E1 -24558.194,E2 -24558.194} C_VEL
LIN {X 0,Y 133.922,Z 612.276,A -85,B 0,C 180,E1 -24560.516,E2 -24560.516} C_VEL
LIN {X 0,Y 133.747,Z 612.847,A -85,B 0,C 180,E1 -24561.321,E2 -24561.321} C_VEL
LIN {X 0,Y 133.571,Z 616.288,A -85,B 0,C 180,E1 -24566.981,E2 -24566.981} C_VEL
LIN {X 0,Y 133.72,Z 617.594,A -85,B 0,C 180,E1 -24569.997,E2 -24569.997} C_VEL
LIN {X 0,Y 133.568,Z 618.522,A -85,B 0,C 180,E1 -24573.013,E2 -24573.013} C_VEL
LIN {X 0,Y 133.759,Z 619.368,A -85,B 0,C 180,E1 -24579.066,E2 -24579.066} C_VEL
LIN {X 0,Y 135.03,Z 618.912,A -85,B 0,C 180,E1 -24585.081,E2 -24585.081} C_VEL
LIN {X 0,Y 137.743,Z 617.179,A -85,B 0,C 180,E1 -24590.923,E2 -24590.923} C_VEL
LIN {X 0,Y 142.148,Z 613.721,A -85,B 0,C 180,E1 -24597.132,E2 -24597.132} C_VEL
LIN {X 0,Y 146.966,Z 609.689,A -85,B 0,C 180,E1 -24601.734,E2 -24601.734} C_VEL
LIN {X 0,Y 153.488,Z 603.727,A -85,B 0,C 180,E1 -24606.527,E2 -24606.527} C_VEL
LIN {X 0,Y 160.042,Z 597.076,A -85,B 0,C 180,E1 -24610.367,E2 -24610.367} C_VEL
LIN {X 0,Y 167.413,Z 588.852,A -85,B 0,C 180,E1 -24613.838,E2 -24613.838} C_VEL
LIN {X 0,Y 174.062,Z 580.34,A -85,B 0,C 180,E1 -24616.613,E2 -24616.613} C_VEL
LIN {X 0,Y 181.221,Z 570.06,A -85,B 0,C 180,E1 -24619.13,E2 -24619.13} C_VEL
LIN {X 0,Y 188.119,Z 558.615,A -85,B 0,C 180,E1 -24621.246,E2 -24621.246} C_VEL
LIN {X 0,Y 193.933,Z 547.257,A -85,B 0,C 180,E1 -24622.866,E2 -24622.866} C_VEL
LIN {X 0,Y 199.36,Z 534.817,A -85,B 0,C 180,E1 -24624.172,E2 -24624.172} C_VEL
LIN {X 0,Y 203.747,Z 522.117,A -85,B 0,C 180,E1 -24625.22,E2 -24625.22} C_VEL
LIN {X 0,Y 207.584,Z 507.969,A -85,B 0,C 180,E1 -24626.02,E2 -24626.02} C_VEL
LIN {X 0,Y 210.251,Z 493.313,A -85,B 0,C 180,E1 -24626.618,E2 -24626.618} C_VEL
LIN {X 0,Y 213.555,Z 459.268,A -85,B 0,C 180,E1 -24627.566,E2 -24627.566} C_VEL
LIN {X 0,Y 210.467,Z 451.079,A -85,B 0,C 180,E1 -24630.165,E2 -24630.165} C_VEL
LIN {X 0,Y 207.646,Z 444.078,A -85,B 0,C 180,E1 -24632.904,E2 -24632.904} C_VEL
LIN {X 0,Y 204.725,Z 437.424,A -85,B 0,C 180,E1 -24636.233,E2 -24636.233} C_VEL
LIN {X 0,Y 202.507,Z 432.921,A -85,B 0,C 180,E1 -24639.305,E2 -24639.305} C_VEL
LIN {X 0,Y 200.527,Z 428.651,A -85,B 0,C 180,E1 -24643.217,E2 -24643.217} C_VEL
LIN {X 0,Y 198.765,Z 425.854,A -85,B 0,C 180,E1 -24650.887,E2 -24650.887} C_VEL
LIN {X 0,Y 198.804,Z 426.047,A -85,B 0,C 180,E1 -24652.638,E2 -24652.638} C_VEL
LIN {X 0,Y 200.618,Z 428.318,A -85,B 0,C 180,E1 -24659.435,E2 -24659.435} C_VEL
LIN {X 0,Y 202.656,Z 432.227,A -85,B 0,C 180,E1 -24663.339,E2 -24663.339} C_VEL
LIN {X 0,Y 203.451,Z 433.672,A -85,B 0,C 180,E1 -24664.489,E2 -24664.489} C_VEL
LIN {X 0,Y 205.835,Z 437.731,A -85,B 0,C 180,E1 -24667.415,E2 -24667.415} C_VEL
LIN {X 0,Y 208.264,Z 442.102,A -85,B 0,C 180,E1 -24669.932,E2 -24669.932} C_VEL
LIN {X 0,Y 211.593,Z 448.402,A -85,B 0,C 180,E1 -24672.898,E2 -24672.898} C_VEL
LIN {X 0,Y 214.022,Z 453.275,A -85,B 0,C 180,E1 -24674.789,E2 -24674.789} C_VEL
LIN {X 0,Y 210.706,Z 487.14,A -85,B 0,C 180,E1 -24675.755,E2 -24675.755} C_VEL
LIN {X 0,Y 208.263,Z 500.782,A -85,B 0,C 180,E1 -24676.351,E2 -24676.351} C_VEL
LIN {X 0,Y 204.666,Z 514.791,A -85,B 0,C 180,E1 -24677.253,E2 -24677.253} C_VEL
LIN {X 0,Y 200.068,Z 528.441,A -85,B 0,C 180,E1 -24678.483,E2 -24678.483} C_VEL
LIN {X 0,Y 194.536,Z 541.557,A -85,B 0,C 180,E1 -24680.072,E2 -24680.072} C_VEL
LIN {X 0,Y 188.41,Z 553.34,A -85,B 0,C 180,E1 -24681.901,E2 -24681.901} C_VEL
LIN {X 0,Y 182.512,Z 563.092,A -85,B 0,C 180,E1 -24683.865,E2 -24683.865} C_VEL
LIN {X 0,Y 175.297,Z 573.381,A -85,B 0,C 180,E1 -24686.54,E2 -24686.54} C_VEL
LIN {X 0,Y 169.043,Z 581.235,A -85,B 0,C 180,E1 -24689.187,E2 -24689.187} C_VEL
LIN {X 0,Y 161.327,Z 589.73,A -85,B 0,C 180,E1 -24693.012,E2 -24693.012} C_VEL
LIN {X 0,Y 154.413,Z 596.456,A -85,B 0,C 180,E1 -24697.207,E2 -24697.207} C_VEL
LIN {X 0,Y 148.818,Z 601.293,A -85,B 0,C 180,E1 -24701.387,E2 -24701.387} C_VEL
LIN {X 0,Y 143.313,Z 605.471,A -85,B 0,C 180,E1 -24706.646,E2 -24706.646} C_VEL
LIN {X 0,Y 138.775,Z 608.313,A -85,B 0,C 180,E1 -24712.579,E2 -24712.579} C_VEL
LIN {X 0,Y 135.614,Z 609.614,A -85,B 0,C 180,E1 -24718.79,E2 -24718.79} C_VEL
LIN {X 0,Y 133.801,Z 609.402,A -85,B 0,C 180,E1 -24725.156,E2 -24725.156} C_VEL
LIN {X 0,Y 133.112,Z 607.746,A -85,B 0,C 180,E1 -24731.534,E2 -24731.534} C_VEL
LIN {X 0,Y 133.162,Z 606.379,A -85,B 0,C 180,E1 -24734.702,E2 -24734.702} C_VEL
LIN {X 0,Y 134.02,Z 602.542,A -85,B 0,C 180,E1 -24740.951,E2 -24740.951} C_VEL
LIN {X 0,Y 135.191,Z 598.638,A -85,B 0,C 180,E1 -24745.53,E2 -24745.53} C_VEL
LIN {X 0,Y 136.874,Z 593.819,A -85,B 0,C 180,E1 -24750.003,E2 -24750.003} C_VEL
LIN {X 0,Y 139.669,Z 586.819,A -85,B 0,C 180,E1 -24755.054,E2 -24755.054} C_VEL
LIN {X 0,Y 142.565,Z 579.872,A -85,B 0,C 180,E1 -24759.037,E2 -24759.037} C_VEL
LIN {X 0,Y 146.35,Z 570.729,A -85,B 0,C 180,E1 -24763.188,E2 -24763.188} C_VEL
LIN {X 0,Y 150.552,Z 560.079,A -85,B 0,C 180,E1 -24766.966,E2 -24766.966} C_VEL
LIN {X 0,Y 154.557,Z 549.307,A -85,B 0,C 180,E1 -24769.942,E2 -24769.942} C_VEL
LIN {X 0,Y 158.473,Z 537.536,A -85,B 0,C 180,E1 -24772.491,E2 -24772.491} C_VEL
LIN {X 0,Y 162.166,Z 524.423,A -85,B 0,C 180,E1 -24774.691,E2 -24774.691} C_VEL
LIN {X 0,Y 165.263,Z 510.917,A -85,B 0,C 180,E1 -24776.391,E2 -24776.391} C_VEL
LIN {X 0,Y 167.63,Z 496.803,A -85,B 0,C 180,E1 -24777.685,E2 -24777.685} C_VEL
LIN {X 0,Y 169.347,Z 482.42,A -85,B 0,C 180,E1 -24778.526,E2 -24778.526} C_VEL
LIN {X 0,Y 173.561,Z 423.205,A -85,B 0,C 180,E1 -24780.663,E2 -24780.663} C_VEL
LIN {X 0,Y 172.606,Z 420.525,A -85,B 0,C 180,E1 -24781.095,E2 -24781.095} C_VEL
LIN {X 0,Y 166.35,Z 407.489,A -85,B 0,C 180,E1 -24783.85,E2 -24783.85} C_VEL
LIN {X 0,Y 159.917,Z 396.016,A -85,B 0,C 180,E1 -24786.944,E2 -24786.944} C_VEL
LIN {X 0,Y 154.668,Z 387.717,A -85,B 0,C 180,E1 -24789.739,E2 -24789.739} C_VEL
LIN {X 0,Y 150.195,Z 381.234,A -85,B 0,C 180,E1 -24792.372,E2 -24792.372} C_VEL
LIN {X 0,Y 147.224,Z 377.207,A -85,B 0,C 180,E1 -24794.272,E2 -24794.272} C_VEL
LIN {X 0,Y 144.647,Z 373.789,A -85,B 0,C 180,E1 -24796.041,E2 -24796.041} C_VEL
LIN {X 0,Y 143.876,Z 372.734,A -85,B 0,C 180,E1 -24796.601,E2 -24796.601} C_VEL
LIN {X 0,Y 141.395,Z 370.092,A -85,B 0,C 180,E1 -24798.434,E2 -24798.434} C_VEL
LIN {X 0,Y 140.157,Z 367.748,A -85,B 0,C 180,E1 -24799.517,E2 -24799.517} C_VEL
LIN {X 0,Y 137.772,Z 365.977,A -85,B 0,C 180,E1 -24801.456,E2 -24801.456} C_VEL
LIN {X 0,Y 136.371,Z 363.56,A -85,B 0,C 180,E1 -24802.849,E2 -24802.849} C_VEL
LIN {X 0,Y 136.029,Z 362.113,A -85,B 0,C 180,E1 -24803.376,E2 -24803.376} C_VEL
LIN {X 0,Y 136.056,Z 362.16,A -85,B 0,C 180,E1 -24808.9,E2 -24808.9} C_VEL
LIN {X 0,Y 136.121,Z 362.14,A -85,B 0,C 180,E1 -24812.312,E2 -24812.312} C_VEL
LIN {X 0,Y 136.188,Z 362.132,A -85,B 0,C 180,E1 -24818.825,E2 -24818.825} C_VEL
LIN {X 0,Y 136.226,Z 362.094,A -85,B 0,C 180,E1 -24825.052,E2 -24825.052} C_VEL
LIN {X 0,Y 136.43,Z 362.055,A -85,B 0,C 180,E1 -24828.18,E2 -24828.18} C_VEL
LIN {X 0,Y 136.55,Z 362.073,A -85,B 0,C 180,E1 -24831.119,E2 -24831.119} C_VEL
LIN {X 0,Y 137.124,Z 361.971,A -85,B 0,C 180,E1 -24840.001,E2 -24840.001} C_VEL
LIN {X 0,Y 136.545,Z 362.089,A -85,B 0,C 180,E1 -24848.884,E2 -24848.884} C_VEL
LIN {X 0,Y 136.447,Z 362.112,A -85,B 0,C 180,E1 -24851.891,E2 -24851.891} C_VEL
LIN {X 0,Y 136.216,Z 362.131,A -85,B 0,C 180,E1 -24858.326,E2 -24858.326} C_VEL
LIN {X 0,Y 136.945,Z 364.469,A -85,B 0,C 180,E1 -24859.195,E2 -24859.195} C_VEL
LIN {X 0,Y 139.119,Z 367.002,A -85,B 0,C 180,E1 -24861.132,E2 -24861.132} C_VEL
LIN {X 0,Y 140.442,Z 367.908,A -85,B 0,C 180,E1 -24862.164,E2 -24862.164} C_VEL
LIN {X 0,Y 142.132,Z 370.935,A -85,B 0,C 180,E1 -24863.592,E2 -24863.592} C_VEL
LIN {X 0,Y 144.504,Z 373.282,A -85,B 0,C 180,E1 -24865.283,E2 -24865.283} C_VEL
LIN {X 0,Y 146.884,Z 376.788,A -85,B 0,C 180,E1 -24866.974,E2 -24866.974} C_VEL
LIN {X 0,Y 148.303,Z 378.447,A -85,B 0,C 180,E1 -24867.888,E2 -24867.888} C_VEL
LIN {X 0,Y 152.356,Z 384.335,A -85,B 0,C 180,E1 -24870.397,E2 -24870.397} C_VEL
LIN {X 0,Y 156.588,Z 390.646,A -85,B 0,C 180,E1 -24872.779,E2 -24872.779} C_VEL
LIN {X 0,Y 159.427,Z 395.578,A -85,B 0,C 180,E1 -24874.295,E2 -24874.295} C_VEL
LIN {X 0,Y 164.768,Z 407.249,A -85,B 0,C 180,E1 -24877.049,E2 -24877.049} C_VEL
LIN {X 0,Y 170.469,Z 422.213,A -85,B 0,C 180,E1 -24879.816,E2 -24879.816} C_VEL
LIN {X 0,Y 173.179,Z 430.499,A -85,B 0,C 180,E1 -24881.102,E2 -24881.102} C_VEL
LIN {X 0,Y 168.71,Z 494.696,A -85,B 0,C 180,E1 -24883.484,E2 -24883.484} C_VEL
LIN {X 0,Y 166.829,Z 508.781,A -85,B 0,C 180,E1 -24884.367,E2 -24884.367} C_VEL
LIN {X 0,Y 164.148,Z 522.944,A -85,B 0,C 180,E1 -24885.697,E2 -24885.697} C_VEL
LIN {X 0,Y 160.784,Z 536.034,A -85,B 0,C 180,E1 -24887.348,E2 -24887.348} C_VEL
LIN {X 0,Y 157.277,Z 547.892,A -85,B 0,C 180,E1 -24889.354,E2 -24889.354} C_VEL
LIN {X 0,Y 154.385,Z 556.824,A -85,B 0,C 180,E1 -24891.247,E2 -24891.247} C_VEL
LIN {X 0,Y 150.587,Z 567.053,A -85,B 0,C 180,E1 -24893.896,E2 -24893.896} C_VEL
LIN {X 0,Y 146.341,Z 577.442,A -85,B 0,C 180,E1 -24897.295,E2 -24897.295} C_VEL
LIN {X 0,Y 142.526,Z 586.846,A -85,B 0,C 180,E1 -24901.261,E2 -24901.261} C_VEL
LIN {X 0,Y 139.117,Z 595.044,A -85,B 0,C 180,E1 -24905.645,E2 -24905.645} C_VEL
LIN {X 0,Y 136.556,Z 602.078,A -85,B 0,C 180,E1 -24910.453,E2 -24910.453} C_VEL
LIN {X 0,Y 134.867,Z 607.254,A -85,B 0,C 180,E1 -24914.895,E2 -24914.895} C_VEL
LIN {X 0,Y 133.948,Z 611.383,A -85,B 0,C 180,E1 -24919.416,E2 -24919.416} C_VEL
LIN {X 0,Y 133.747,Z 612.847,A -85,B 0,C 180,E1 -24921.321,E2 -24921.321} C_VEL
LIN {X 0,Y 132.896,Z 614.466,A -85,B 0,C 180,E1 -24923.743,E2 -24923.743} C_VEL
LIN {X 0,Y 131.244,Z 615.781,A -85,B 0,C 180,E1 -24926.16,E2 -24926.16} C_VEL
LIN {X 0,Y 127.542,Z 617.647,A -85,B 0,C 180,E1 -24931.175,E2 -24931.175} C_VEL
LIN {X 0,Y 126.421,Z 618.46,A -85,B 0,C 180,E1 -24934.745,E2 -24934.745} C_VEL
LIN {X 0,Y 126.724,Z 619.077,A -85,B 0,C 180,E1 -24939.574,E2 -24939.574} C_VEL
LIN {X 0,Y 128.133,Z 618.704,A -85,B 0,C 180,E1 -24945.914,E2 -24945.914} C_VEL
LIN {X 0,Y 131.078,Z 617.055,A -85,B 0,C 180,E1 -24952.041,E2 -24952.041} C_VEL
LIN {X 0,Y 135.519,Z 613.91,A -85,B 0,C 180,E1 -24958.16,E2 -24958.16} C_VEL
LIN {X 0,Y 140.957,Z 609.745,A -85,B 0,C 180,E1 -24963.257,E2 -24963.257} C_VEL
LIN {X 0,Y 147.835,Z 603.882,A -85,B 0,C 180,E1 -24968.168,E2 -24968.168} C_VEL
LIN {X 0,Y 154.715,Z 597.336,A -85,B 0,C 180,E1 -24972.065,E2 -24972.065} C_VEL
LIN {X 0,Y 162.39,Z 589.265,A -85,B 0,C 180,E1 -24975.566,E2 -24975.566} C_VEL
LIN {X 0,Y 169.784,Z 580.261,A -85,B 0,C 180,E1 -24978.524,E2 -24978.524} C_VEL
LIN {X 0,Y 176.694,Z 570.796,A -85,B 0,C 180,E1 -24980.857,E2 -24980.857} C_VEL
LIN {X 0,Y 183.793,Z 559.566,A -85,B 0,C 180,E1 -24982.957,E2 -24982.957} C_VEL
LIN {X 0,Y 189.781,Z 548.465,A -85,B 0,C 180,E1 -24984.555,E2 -24984.555} C_VEL
LIN {X 0,Y 195.341,Z 536.374,A -85,B 0,C 180,E1 -24985.838,E2 -24985.838} C_VEL
LIN {X 0,Y 200.187,Z 523.067,A -85,B 0,C 180,E1 -24986.945,E2 -24986.945} C_VEL
LIN {X 0,Y 204.289,Z 508.587,A -85,B 0,C 180,E1 -24987.762,E2 -24987.762} C_VEL
LIN {X 0,Y 207.066,Z 494.124,A -85,B 0,C 180,E1 -24988.352,E2 -24988.352} C_VEL
LIN {X 0,Y 210.246,Z 463.409,A -85,B 0,C 180,E1 -24989.201,E2 -24989.201} C_VEL
LIN {X 0,Y 210.243,Z 462.325,A -85,B 0,C 180,E1 -24989.298,E2 -24989.298} C_VEL
LIN {X 0,Y 207.238,Z 453.925,A -85,B 0,C 180,E1 -24992.196,E2 -24992.196} C_VEL
LIN {X 0,Y 204.705,Z 447.633,A -85,B 0,C 180,E1 -24994.984,E2 -24994.984} C_VEL
LIN {X 0,Y 202.992,Z 443.548,A -85,B 0,C 180,E1 -24997.175,E2 -24997.175} C_VEL
LIN {X 0,Y 201.088,Z 439.4,A -85,B 0,C 180,E1 -25000.054,E2 -25000.054} C_VEL
LIN {X 0,Y 199.438,Z 435.566,A -85,B 0,C 180,E1 -25003.625,E2 -25003.625} C_VEL
LIN {X 0,Y 197.871,Z 432.929,A -85,B 0,C 180,E1 -25010.846,E2 -25010.846} C_VEL
LIN {X 0,Y 197.905,Z 433.091,A -85,B 0,C 180,E1 -25012.571,E2 -25012.571} C_VEL
LIN {X 0,Y 199.567,Z 435.311,A -85,B 0,C 180,E1 -25019.127,E2 -25019.127} C_VEL
LIN {X 0,Y 201.445,Z 439.07,A -85,B 0,C 180,E1 -25022.931,E2 -25022.931} C_VEL
LIN {X 0,Y 204.284,Z 444.25,A -85,B 0,C 180,E1 -25026.774,E2 -25026.774} C_VEL
LIN {X 0,Y 207.44,Z 450.222,A -85,B 0,C 180,E1 -25030.138,E2 -25030.138} C_VEL
LIN {X 0,Y 210.784,Z 457.14,A -85,B 0,C 180,E1 -25033.151,E2 -25033.151} C_VEL
LIN {X 0,Y 207.625,Z 487.732,A -85,B 0,C 180,E1 -25034.011,E2 -25034.011} C_VEL
LIN {X 0,Y 205.041,Z 501.549,A -85,B 0,C 180,E1 -25034.609,E2 -25034.609} C_VEL
LIN {X 0,Y 201.438,Z 515.114,A -85,B 0,C 180,E1 -25035.469,E2 -25035.469} C_VEL
LIN {X 0,Y 196.668,Z 528.83,A -85,B 0,C 180,E1 -25036.68,E2 -25036.68} C_VEL
LIN {X 0,Y 191.338,Z 541.095,A -85,B 0,C 180,E1 -25038.127,E2 -25038.127} C_VEL
LIN {X 0,Y 185.165,Z 552.778,A -85,B 0,C 180,E1 -25039.891,E2 -25039.891} C_VEL
LIN {X 0,Y 178.227,Z 563.877,A -85,B 0,C 180,E1 -25042.085,E2 -25042.085} C_VEL
LIN {X 0,Y 171.21,Z 573.485,A -85,B 0,C 180,E1 -25044.568,E2 -25044.568} C_VEL
LIN {X 0,Y 164.336,Z 581.746,A -85,B 0,C 180,E1 -25047.353,E2 -25047.353} C_VEL
LIN {X 0,Y 157.273,Z 589.214,A -85,B 0,C 180,E1 -25050.664,E2 -25050.664} C_VEL
LIN {X 0,Y 151.624,Z 594.554,A -85,B 0,C 180,E1 -25053.794,E2 -25053.794} C_VEL
LIN {X 0,Y 146.027,Z 599.324,A -85,B 0,C 180,E1 -25057.433,E2 -25057.433} C_VEL
LIN {X 0,Y 139.3,Z 604.418,A -85,B 0,C 180,E1 -25062.987,E2 -25062.987} C_VEL
LIN {X 0,Y 135.114,Z 607.087,A -85,B 0,C 180,E1 -25067.457,E2 -25067.457} C_VEL
LIN {X 0,Y 130.793,Z 609.285,A -85,B 0,C 180,E1 -25073.771,E2 -25073.771} C_VEL
LIN {X 0,Y 127.882,Z 609.987,A -85,B 0,C 180,E1 -25080.359,E2 -25080.359} C_VEL
LIN {X 0,Y 126.367,Z 609.193,A -85,B 0,C 180,E1 -25087.092,E2 -25087.092} C_VEL
LIN {X 0,Y 126.013,Z 606.944,A -85,B 0,C 180,E1 -25093.811,E2 -25093.811} C_VEL
LIN {X 0,Y 126.805,Z 603.232,A -85,B 0,C 180,E1 -25100.432,E2 -25100.432} C_VEL
LIN {X 0,Y 127.976,Z 599.463,A -85,B 0,C 180,E1 -25105.278,E2 -25105.278} C_VEL
LIN {X 0,Y 129.662,Z 594.767,A -85,B 0,C 180,E1 -25110.003,E2 -25110.003} C_VEL
LIN {X 0,Y 132.499,Z 587.947,A -85,B 0,C 180,E1 -25115.329,E2 -25115.329} C_VEL
LIN {X 0,Y 135.788,Z 580.441,A -85,B 0,C 180,E1 -25119.894,E2 -25119.894} C_VEL
LIN {X 0,Y 139.395,Z 572.214,A -85,B 0,C 180,E1 -25123.859,E2 -25123.859} C_VEL
LIN {X 0,Y 143.719,Z 561.829,A -85,B 0,C 180,E1 -25127.799,E2 -25127.799} C_VEL
LIN {X 0,Y 148.284,Z 550.165,A -85,B 0,C 180,E1 -25131.188,E2 -25131.188} C_VEL
LIN {X 0,Y 152.373,Z 538.508,A -85,B 0,C 180,E1 -25133.805,E2 -25133.805} C_VEL
LIN {X 0,Y 156.176,Z 525.728,A -85,B 0,C 180,E1 -25136.027,E2 -25136.027} C_VEL
LIN {X 0,Y 159.221,Z 513.02,A -85,B 0,C 180,E1 -25137.719,E2 -25137.719} C_VEL
LIN {X 0,Y 161.759,Z 499.376,A -85,B 0,C 180,E1 -25139.053,E2 -25139.053} C_VEL
LIN {X 0,Y 163.673,Z 485.315,A -85,B 0,C 180,E1 -25139.962,E2 -25139.962} C_VEL
LIN {X 0,Y 168.094,Z 424.843,A -85,B 0,C 180,E1 -25142.234,E2 -25142.234} C_VEL
LIN {X 0,Y 162.007,Z 411.81,A -85,B 0,C 180,E1 -25145.109,E2 -25145.109} C_VEL
LIN {X 0,Y 156.161,Z 401.055,A -85,B 0,C 180,E1 -25148.124,E2 -25148.124} C_VEL
LIN {X 0,Y 150.147,Z 391.283,A -85,B 0,C 180,E1 -25151.599,E2 -25151.599} C_VEL
LIN {X 0,Y 144.532,Z 383.268,A -85,B 0,C 180,E1 -25155.261,E2 -25155.261} C_VEL
LIN {X 0,Y 141.658,Z 379.318,A -85,B 0,C 180,E1 -25157.368,E2 -25157.368} C_VEL
LIN {X 0,Y 138.703,Z 375.867,A -85,B 0,C 180,E1 -25159.702,E2 -25159.702} C_VEL
LIN {X 0,Y 137.677,Z 374.091,A -85,B 0,C 180,E1 -25160.638,E2 -25160.638} C_VEL
LIN {X 0,Y 135.218,Z 371.821,A -85,B 0,C 180,E1 -25162.829,E2 -25162.829} C_VEL
LIN {X 0,Y 133.575,Z 368.752,A -85,B 0,C 180,E1 -25164.638,E2 -25164.638} C_VEL
LIN {X 0,Y 130.87,Z 367.043,A -85,B 0,C 180,E1 -25167.52,E2 -25167.52} C_VEL
LIN {X 0,Y 129.351,Z 364.498,A -85,B 0,C 180,E1 -25169.605,E2 -25169.605} C_VEL
LIN {X 0,Y 129.01,Z 363.036,A -85,B 0,C 180,E1 -25170.305,E2 -25170.305} C_VEL
LIN {X 0,Y 128.98,Z 363.037,A -85,B 0,C 180,E1 -25174.158,E2 -25174.158} C_VEL
LIN {X 0,Y 129.072,Z 363.018,A -85,B 0,C 180,E1 -25177.773,E2 -25177.773} C_VEL
LIN {X 0,Y 129.149,Z 362.985,A -85,B 0,C 180,E1 -25184.213,E2 -25184.213} C_VEL
LIN {X 0,Y 129.347,Z 362.934,A -85,B 0,C 180,E1 -25187.976,E2 -25187.976} C_VEL
LIN {X 0,Y 129.473,Z 362.942,A -85,B 0,C 180,E1 -25190.629,E2 -25190.629} C_VEL
LIN {X 0,Y 130.079,Z 362.846,A -85,B 0,C 180,E1 -25200.001,E2 -25200.001} C_VEL
LIN {X 0,Y 129.471,Z 362.971,A -85,B 0,C 180,E1 -25209.373,E2 -25209.373} C_VEL
LIN {X 0,Y 129.409,Z 363.052,A -85,B 0,C 180,E1 -25211.683,E2 -25211.683} C_VEL
LIN {X 0,Y 130.101,Z 365.497,A -85,B 0,C 180,E1 -25212.876,E2 -25212.876} C_VEL
LIN {X 0,Y 131.857,Z 367.697,A -85,B 0,C 180,E1 -25215.061,E2 -25215.061} C_VEL
LIN {X 0,Y 133.912,Z 368.975,A -85,B 0,C 180,E1 -25217.171,E2 -25217.171} C_VEL
LIN {X 0,Y 135.532,Z 371.919,A -85,B 0,C 180,E1 -25218.912,E2 -25218.912} C_VEL
LIN {X 0,Y 138.074,Z 374.518,A -85,B 0,C 180,E1 -25221.168,E2 -25221.168} C_VEL
LIN {X 0,Y 140.379,Z 377.906,A -85,B 0,C 180,E1 -25223.125,E2 -25223.125} C_VEL
LIN {X 0,Y 141.945,Z 379.624,A -85,B 0,C 180,E1 -25224.304,E2 -25224.304} C_VEL
LIN {X 0,Y 144.795,Z 383.467,A -85,B 0,C 180,E1 -25226.367,E2 -25226.367} C_VEL
LIN {X 0,Y 148.687,Z 389.196,A -85,B 0,C 180,E1 -25228.968,E2 -25228.968} C_VEL
LIN {X 0,Y 153.226,Z 396.21,A -85,B 0,C 180,E1 -25231.705,E2 -25231.705} C_VEL
LIN {X 0,Y 155.697,Z 400.784,A -85,B 0,C 180,E1 -25233.123,E2 -25233.123} C_VEL
LIN {X 0,Y 160.627,Z 411.981,A -85,B 0,C 180,E1 -25235.855,E2 -25235.855} C_VEL
LIN {X 0,Y 165.892,Z 426.296,A -85,B 0,C 180,E1 -25238.602,E2 -25238.602} C_VEL
LIN {X 0,Y 167.797,Z 432.34,A -85,B 0,C 180,E1 -25239.574,E2 -25239.574} C_VEL
LIN {X 0,Y 163.313,Z 494.169,A -85,B 0,C 180,E1 -25241.893,E2 -25241.893} C_VEL
LIN {X 0,Y 161.334,Z 508.484,A -85,B 0,C 180,E1 -25242.796,E2 -25242.796} C_VEL
LIN {X 0,Y 158.563,Z 522.671,A -85,B 0,C 180,E1 -25244.15,E2 -25244.15} C_VEL
LIN {X 0,Y 155.062,Z 535.761,A -85,B 0,C 180,E1 -25245.822,E2 -25245.822} C_VEL
LIN {X 0,Y 151.087,Z 548.576,A -85,B 0,C 180,E1 -25248.053,E2 -25248.053} C_VEL
LIN {X 0,Y 146.99,Z 560.136,A -85,B 0,C 180,E1 -25250.687,E2 -25250.687} C_VEL
LIN {X 0,Y 142.767,Z 570.785,A -85,B 0,C 180,E1 -25253.789,E2 -25253.789} C_VEL
LIN {X 0,Y 138.2,Z 581.337,A -85,B 0,C 180,E1 -25257.724,E2 -25257.724} C_VEL
LIN {X 0,Y 134.479,Z 590.044,A -85,B 0,C 180,E1 -25261.94,E2 -25261.94} C_VEL
LIN {X 0,Y 131.021,Z 598.32,A -85,B 0,C 180,E1 -25267.112,E2 -25267.112} C_VEL
LIN {X 0,Y 128.52,Z 604.955,A -85,B 0,C 180,E1 -25272.494,E2 -25272.494} C_VEL
LIN {X 0,Y 126.936,Z 610.81,A -85,B 0,C 180,E1 -25278.824,E2 -25278.824} C_VEL
LIN {X 0,Y 126.535,Z 614.134,A -85,B 0,C 180,E1 -25283.619,E2 -25283.619} C_VEL
LIN {X 0,Y 126.635,Z 617.189,A -85,B 0,C 180,E1 -25289.997,E2 -25289.997} C_VEL
LIN {X 0,Y 126.421,Z 618.46,A -85,B 0,C 180,E1 -25294.745,E2 -25294.745} C_VEL
LIN {X 0,Y 125.809,Z 618.887,A -85,B 0,C 180,E1 -25297.407,E2 -25297.407} C_VEL
LIN {X 0,Y 123.471,Z 618.985,A -85,B 0,C 180,E1 -25301.841,E2 -25301.841} C_VEL
LIN {X 0,Y 121.953,Z 618.696,A -85,B 0,C 180,E1 -25305.496,E2 -25305.496} C_VEL
LIN {X 0,Y 121.931,Z 618.261,A -85,B 0,C 180,E1 -25308.279,E2 -25308.279} C_VEL
LIN {X 0,Y 122.254,Z 618.049,A -85,B 0,C 180,E1 -25309.192,E2 -25309.192} C_VEL
LIN {X 0,Y 124.47,Z 616.932,A -85,B 0,C 180,E1 -25313.278,E2 -25313.278} C_VEL
LIN {X 0,Y 128.985,Z 614.059,A -85,B 0,C 180,E1 -25319.362,E2 -25319.362} C_VEL
LIN {X 0,Y 135.047,Z 609.801,A -85,B 0,C 180,E1 -25324.918,E2 -25324.918} C_VEL
LIN {X 0,Y 142.298,Z 604.036,A -85,B 0,C 180,E1 -25329.942,E2 -25329.942} C_VEL
LIN {X 0,Y 149.533,Z 597.594,A -85,B 0,C 180,E1 -25333.884,E2 -25333.884} C_VEL
LIN {X 0,Y 157.508,Z 589.641,A -85,B 0,C 180,E1 -25337.407,E2 -25337.407} C_VEL
LIN {X 0,Y 164.667,Z 581.379,A -85,B 0,C 180,E1 -25340.192,E2 -25340.192} C_VEL
LIN {X 0,Y 172.335,Z 571.464,A -85,B 0,C 180,E1 -25342.673,E2 -25342.673} C_VEL
LIN {X 0,Y 179.646,Z 560.481,A -85,B 0,C 180,E1 -25344.748,E2 -25344.748} C_VEL
LIN {X 0,Y 186.489,Z 548.298,A -85,B 0,C 180,E1 -25346.487,E2 -25346.487} C_VEL
LIN {X 0,Y 192.206,Z 536.258,A -85,B 0,C 180,E1 -25347.728,E2 -25347.728} C_VEL
LIN {X 0,Y 197.189,Z 523.026,A -85,B 0,C 180,E1 -25348.798,E2 -25348.798} C_VEL
LIN {X 0,Y 201.244,Z 509.185,A -85,B 0,C 180,E1 -25349.571,E2 -25349.571} C_VEL
LIN {X 0,Y 204.145,Z 494.898,A -85,B 0,C 180,E1 -25350.147,E2 -25350.147} C_VEL
LIN {X 0,Y 206.738,Z 472.257,A -85,B 0,C 180,E1 -25350.747,E2 -25350.747} C_VEL
LIN {X 0,Y 207.266,Z 465.854,A -85,B 0,C 180,E1 -25350.99,E2 -25350.99} C_VEL
LIN {X 0,Y 204.715,Z 458.375,A -85,B 0,C 180,E1 -25353.733,E2 -25353.733} C_VEL
LIN {X 0,Y 202.768,Z 453.281,A -85,B 0,C 180,E1 -25356.105,E2 -25356.105} C_VEL
LIN {X 0,Y 201.437,Z 449.928,A -85,B 0,C 180,E1 -25357.958,E2 -25357.958} C_VEL
LIN {X 0,Y 199.678,Z 445.74,A -85,B 0,C 180,E1 -25360.918,E2 -25360.918} C_VEL
LIN {X 0,Y 198.356,Z 442.44,A -85,B 0,C 180,E1 -25364.059,E2 -25364.059} C_VEL
LIN {X 0,Y 196.99,Z 439.87,A -85,B 0,C 180,E1 -25371.795,E2 -25371.795} C_VEL
LIN {X 0,Y 198.486,Z 442.201,A -85,B 0,C 180,E1 -25378.714,E2 -25378.714} C_VEL
LIN {X 0,Y 200.623,Z 446.765,A -85,B 0,C 180,E1 -25383.158,E2 -25383.158} C_VEL
LIN {X 0,Y 202.857,Z 451.009,A -85,B 0,C 180,E1 -25386.254,E2 -25386.254} C_VEL
LIN {X 0,Y 205.814,Z 456.97,A -85,B 0,C 180,E1 -25389.574,E2 -25389.574} C_VEL
LIN {X 0,Y 207.775,Z 461.281,A -85,B 0,C 180,E1 -25391.492,E2 -25391.492} C_VEL
LIN {X 0,Y 204.898,Z 487.726,A -85,B 0,C 180,E1 -25392.189,E2 -25392.189} C_VEL
LIN {X 0,Y 202.24,Z 501.66,A -85,B 0,C 180,E1 -25392.772,E2 -25392.772} C_VEL
LIN {X 0,Y 198.414,Z 515.625,A -85,B 0,C 180,E1 -25393.634,E2 -25393.634} C_VEL
LIN {X 0,Y 193.638,Z 528.928,A -85,B 0,C 180,E1 -25394.783,E2 -25394.783} C_VEL
LIN {X 0,Y 188.384,Z 540.703,A -85,B 0,C 180,E1 -25396.135,E2 -25396.135} C_VEL
LIN {X 0,Y 182.229,Z 552.097,A -85,B 0,C 180,E1 -25397.796,E2 -25397.796} C_VEL
LIN {X 0,Y 175.5,Z 562.638,A -85,B 0,C 180,E1 -25399.775,E2 -25399.775} C_VEL
LIN {X 0,Y 168.708,Z 571.844,A -85,B 0,C 180,E1 -25402.018,E2 -25402.018} C_VEL
LIN {X 0,Y 160.863,Z 581.095,A -85,B 0,C 180,E1 -25404.973,E2 -25404.973} C_VEL
LIN {X 0,Y 153.517,Z 588.642,A -85,B 0,C 180,E1 -25408.211,E2 -25408.211} C_VEL
LIN {X 0,Y 146.561,Z 594.927,A -85,B 0,C 180,E1 -25411.834,E2 -25411.834} C_VEL
LIN {X 0,Y 139.531,Z 600.534,A -85,B 0,C 180,E1 -25416.308,E2 -25416.308} C_VEL
LIN {X 0,Y 134.168,Z 604.281,A -85,B 0,C 180,E1 -25420.581,E2 -25420.581} C_VEL
LIN {X 0,Y 129.544,Z 607.085,A -85,B 0,C 180,E1 -25425.153,E2 -25425.153} C_VEL
LIN {X 0,Y 124.691,Z 609.414,A -85,B 0,C 180,E1 -25431.688,E2 -25431.688} C_VEL
LIN {X 0,Y 121.321,Z 610.242,A -85,B 0,C 180,E1 -25438.58,E2 -25438.58} C_VEL
LIN {X 0,Y 119.445,Z 609.606,A -85,B 0,C 180,E1 -25445.681,E2 -25445.681} C_VEL
LIN {X 0,Y 118.941,Z 608.159,A -85,B 0,C 180,E1 -25450.978,E2 -25450.978} C_VEL
LIN {X 0,Y 119.035,Z 605.898,A -85,B 0,C 180,E1 -25456.343,E2 -25456.343} C_VEL
LIN {X 0,Y 119.902,Z 602.802,A -85,B 0,C 180,E1 -25461.577,E2 -25461.577} C_VEL
LIN {X 0,Y 121.23,Z 598.807,A -85,B 0,C 180,E1 -25466.68,E2 -25466.68} C_VEL
LIN {X 0,Y 123.162,Z 593.887,A -85,B 0,C 180,E1 -25471.638,E2 -25471.638} C_VEL
LIN {X 0,Y 126.368,Z 586.774,A -85,B 0,C 180,E1 -25477.191,E2 -25477.191} C_VEL
LIN {X 0,Y 129.751,Z 579.485,A -85,B 0,C 180,E1 -25481.643,E2 -25481.643} C_VEL
LIN {X 0,Y 133.873,Z 570.421,A -85,B 0,C 180,E1 -25486.001,E2 -25486.001} C_VEL
LIN {X 0,Y 138.569,Z 559.598,A -85,B 0,C 180,E1 -25490.023,E2 -25490.023} C_VEL
LIN {X 0,Y 142.996,Z 548.617,A -85,B 0,C 180,E1 -25493.155,E2 -25493.155} C_VEL
LIN {X 0,Y 147.312,Z 536.574,A -85,B 0,C 180,E1 -25495.809,E2 -25495.809} C_VEL
LIN {X 0,Y 151.255,Z 523.357,A -85,B 0,C 180,E1 -25498.046,E2 -25498.046} C_VEL
LIN {X 0,Y 154.551,Z 509.55,A -85,B 0,C 180,E1 -25499.763,E2 -25499.763} C_VEL
LIN {X 0,Y 157.008,Z 495.664,A -85,B 0,C 180,E1 -25501.005,E2 -25501.005} C_VEL
LIN {X 0,Y 158.776,Z 480.694,A -85,B 0,C 180,E1 -25501.86,E2 -25501.86} C_VEL
LIN {X 0,Y 162.829,Z 427.191,A -85,B 0,C 180,E1 -25503.841,E2 -25503.841} C_VEL
LIN {X 0,Y 157.219,Z 415.07,A -85,B 0,C 180,E1 -25506.717,E2 -25506.717} C_VEL
LIN {X 0,Y 151.809,Z 405.007,A -85,B 0,C 180,E1 -25509.746,E2 -25509.746} C_VEL
LIN {X 0,Y 146.581,Z 396.301,A -85,B 0,C 180,E1 -25513.016,E2 -25513.016} C_VEL
LIN {X 0,Y 141.539,Z 388.972,A -85,B 0,C 180,E1 -25516.53,E2 -25516.53} C_VEL
LIN {X 0,Y 138.422,Z 384.707,A -85,B 0,C 180,E1 -25518.984,E2 -25518.984} C_VEL
LIN {X 0,Y 135.816,Z 381.217,A -85,B 0,C 180,E1 -25521.267,E2 -25521.267} C_VEL
LIN {X 0,Y 135.088,Z 380.26,A -85,B 0,C 180,E1 -25521.949,E2 -25521.949} C_VEL
LIN {X 0,Y 132.478,Z 377.177,A -85,B 0,C 180,E1 -25524.56,E2 -25524.56} C_VEL
LIN {X 0,Y 131.409,Z 375.321,A -85,B 0,C 180,E1 -25525.818,E2 -25525.818} C_VEL
LIN {X 0,Y 128.721,Z 373.098,A -85,B 0,C 180,E1 -25528.985,E2 -25528.985} C_VEL
LIN {X 0,Y 127.003,Z 369.836,A -85,B 0,C 180,E1 -25531.681,E2 -25531.681} C_VEL
LIN {X 0,Y 124.076,Z 368.134,A -85,B 0,C 180,E1 -25536.642,E2 -25536.642} C_VEL
LIN {X 0,Y 122.276,Z 365.103,A -85,B 0,C 180,E1 -25541.79,E2 -25541.79} C_VEL
LIN {X 0,Y 122.063,Z 363.88,A -85,B 0,C 180,E1 -25543.27,E2 -25543.27} C_VEL
LIN {X 0,Y 122.291,Z 363.811,A -85,B 0,C 180,E1 -25547.694,E2 -25547.694} C_VEL
LIN {X 0,Y 122.399,Z 363.813,A -85,B 0,C 180,E1 -25550.082,E2 -25550.082} C_VEL
LIN {X 0,Y 122.568,Z 363.799,A -85,B 0,C 180,E1 -25556.714,E2 -25556.714} C_VEL
LIN {X 0,Y 123.031,Z 363.722,A -85,B 0,C 180,E1 -25560.001,E2 -25560.001} C_VEL
LIN {X 0,Y 122.878,Z 363.824,A -85,B 0,C 180,E1 -25560.923,E2 -25560.923} C_VEL
LIN {X 0,Y 123.234,Z 365.857,A -85,B 0,C 180,E1 -25562.453,E2 -25562.453} C_VEL
LIN {X 0,Y 124.754,Z 368.281,A -85,B 0,C 180,E1 -25566.064,E2 -25566.064} C_VEL
LIN {X 0,Y 127.562,Z 370.029,A -85,B 0,C 180,E1 -25570.554,E2 -25570.554} C_VEL
LIN {X 0,Y 128.858,Z 372.89,A -85,B 0,C 180,E1 -25572.602,E2 -25572.602} C_VEL
LIN {X 0,Y 131.316,Z 375.181,A -85,B 0,C 180,E1 -25575.551,E2 -25575.551} C_VEL
LIN {X 0,Y 131.967,Z 375.853,A -85,B 0,C 180,E1 -25576.267,E2 -25576.267} C_VEL
LIN {X 0,Y 134.328,Z 379.338,A -85,B 0,C 180,E1 -25578.791,E2 -25578.791} C_VEL
LIN {X 0,Y 135.794,Z 380.943,A -85,B 0,C 180,E1 -25580.152,E2 -25580.152} C_VEL
LIN {X 0,Y 138.338,Z 384.52,A -85,B 0,C 180,E1 -25582.402,E2 -25582.402} C_VEL
LIN {X 0,Y 140.027,Z 386.861,A -85,B 0,C 180,E1 -25583.773,E2 -25583.773} C_VEL
LIN {X 0,Y 143.181,Z 391.216,A -85,B 0,C 180,E1 -25586.119,E2 -25586.119} C_VEL
LIN {X 0,Y 147.822,Z 398.337,A -85,B 0,C 180,E1 -25589.263,E2 -25589.263} C_VEL
LIN {X 0,Y 151.427,Z 404.602,A -85,B 0,C 180,E1 -25591.512,E2 -25591.512} C_VEL
LIN {X 0,Y 155.842,Z 414.888,A -85,B 0,C 180,E1 -25594.18,E2 -25594.18} C_VEL
LIN {X 0,Y 160.845,Z 428.843,A -85,B 0,C 180,E1 -25597.026,E2 -25597.026} C_VEL
LIN {X 0,Y 162.538,Z 434.263,A -85,B 0,C 180,E1 -25597.962,E2 -25597.962} C_VEL
LIN {X 0,Y 157.958,Z 494.265,A -85,B 0,C 180,E1 -25600.241,E2 -25600.241} C_VEL
LIN {X 0,Y 155.847,Z 508.826,A -85,B 0,C 180,E1 -25601.187,E2 -25601.187} C_VEL
LIN {X 0,Y 152.801,Z 523.412,A -85,B 0,C 180,E1 -25602.613,E2 -25602.613} C_VEL
LIN {X 0,Y 148.951,Z 537.193,A -85,B 0,C 180,E1 -25604.465,E2 -25604.465} C_VEL
LIN {X 0,Y 144.75,Z 549.885,A -85,B 0,C 180,E1 -25606.788,E2 -25606.788} C_VEL
LIN {X 0,Y 140.535,Z 560.987,A -85,B 0,C 180,E1 -25609.447,E2 -25609.447} C_VEL
LIN {X 0,Y 136.177,Z 571.453,A -85,B 0,C 180,E1 -25612.667,E2 -25612.667} C_VEL
LIN {X 0,Y 131.459,Z 581.804,A -85,B 0,C 180,E1 -25616.769,E2 -25616.769} C_VEL
LIN {X 0,Y 127.526,Z 590.506,A -85,B 0,C 180,E1 -25621.257,E2 -25621.257} C_VEL
LIN {X 0,Y 123.98,Z 598.541,A -85,B 0,C 180,E1 -25626.618,E2 -25626.618} C_VEL
LIN {X 0,Y 121.704,Z 604.258,A -85,B 0,C 180,E1 -25631.479,E2 -25631.479} C_VEL
LIN {X 0,Y 119.948,Z 610.216,A -85,B 0,C 180,E1 -25638.163,E2 -25638.163} C_VEL
LIN {X 0,Y 119.459,Z 613.629,A -85,B 0,C 180,E1 -25643.24,E2 -25643.24} C_VEL
LIN {X 0,Y 119.567,Z 616.774,A -85,B 0,C 180,E1 -25649.997,E2 -25649.997} C_VEL
LIN {X 0,Y 119.357,Z 618.048,A -85,B 0,C 180,E1 -25654.734,E2 -25654.734} C_VEL
LIN {X 0,Y 119.689,Z 618.784,A -85,B 0,C 180,E1 -25660.143,E2 -25660.143} C_VEL
LIN {X 0,Y 121.27,Z 618.496,A -85,B 0,C 180,E1 -25666.841,E2 -25666.841} C_VEL
LIN {X 0,Y 122.254,Z 618.049,A -85,B 0,C 180,E1 -25669.192,E2 -25669.192} C_VEL
LIN {X 0,Y 122.961,Z 617.419,A -85,B 0,C 180,E1 -25671.915,E2 -25671.915} C_VEL
LIN {X 0,Y 122.893,Z 615.92,A -85,B 0,C 180,E1 -25676.485,E2 -25676.485} C_VEL
LIN {X 0,Y 123.571,Z 613.938,A -85,B 0,C 180,E1 -25680.991,E2 -25680.991} C_VEL
LIN {X 0,Y 125.39,Z 612.414,A -85,B 0,C 180,E1 -25683.488,E2 -25683.488} C_VEL
LIN {X 0,Y 131.068,Z 608.604,A -85,B 0,C 180,E1 -25688.067,E2 -25688.067} C_VEL
LIN {X 0,Y 139.001,Z 602.551,A -85,B 0,C 180,E1 -25693.041,E2 -25693.041} C_VEL
LIN {X 0,Y 146.829,Z 595.807,A -85,B 0,C 180,E1 -25696.878,E2 -25696.878} C_VEL
LIN {X 0,Y 155.221,Z 587.484,A -85,B 0,C 180,E1 -25700.324,E2 -25700.324} C_VEL
LIN {X 0,Y 162.858,Z 578.878,A -85,B 0,C 180,E1 -25702.969,E2 -25702.969} C_VEL
LIN {X 0,Y 170.836,Z 568.501,A -85,B 0,C 180,E1 -25705.359,E2 -25705.359} C_VEL
LIN {X 0,Y 177.782,Z 558.086,A -85,B 0,C 180,E1 -25707.141,E2 -25707.141} C_VEL
LIN {X 0,Y 184.163,Z 546.809,A -85,B 0,C 180,E1 -25708.631,E2 -25708.631} C_VEL
LIN {X 0,Y 190.004,Z 534.494,A -85,B 0,C 180,E1 -25709.834,E2 -25709.834} C_VEL
LIN {X 0,Y 194.721,Z 522.092,A -85,B 0,C 180,E1 -25710.769,E2 -25710.769} C_VEL
LIN {X 0,Y 198.865,Z 508.095,A -85,B 0,C 180,E1 -25711.496,E2 -25711.496} C_VEL
LIN {X 0,Y 201.736,Z 493.914,A -85,B 0,C 180,E1 -25712.046,E2 -25712.046} C_VEL
LIN {X 0,Y 204.492,Z 469.488,A -85,B 0,C 180,E1 -25712.703,E2 -25712.703} C_VEL
LIN {X 0,Y 202.162,Z 462.394,A -85,B 0,C 180,E1 -25715.53,E2 -25715.53} C_VEL
LIN {X 0,Y 199.967,Z 456.394,A -85,B 0,C 180,E1 -25718.683,E2 -25718.683} C_VEL
LIN {X 0,Y 198.426,Z 452.381,A -85,B 0,C 180,E1 -25721.545,E2 -25721.545} C_VEL
LIN {X 0,Y 197.278,Z 449.362,A -85,B 0,C 180,E1 -25724.497,E2 -25724.497} C_VEL
LIN {X 0,Y 196.094,Z 446.933,A -85,B 0,C 180,E1 -25731.757,E2 -25731.757} C_VEL
LIN {X 0,Y 197.412,Z 449.109,A -85,B 0,C 180,E1 -25738.296,E2 -25738.296} C_VEL
LIN {X 0,Y 199.3,Z 453.406,A -85,B 0,C 180,E1 -25742.53,E2 -25742.53} C_VEL
LIN {X 0,Y 201.559,Z 457.982,A -85,B 0,C 180,E1 -25745.869,E2 -25745.869} C_VEL
LIN {X 0,Y 204.414,Z 464.071,A -85,B 0,C 180,E1 -25749.211,E2 -25749.211} C_VEL
LIN {X 0,Y 204.867,Z 465.102,A -85,B 0,C 180,E1 -25749.689,E2 -25749.689} C_VEL
LIN {X 0,Y 202.223,Z 488.713,A -85,B 0,C 180,E1 -25750.356,E2 -25750.356} C_VEL
LIN {X 0,Y 199.51,Z 502.37,A -85,B 0,C 180,E1 -25750.92,E2 -25750.92} C_VEL
LIN {X 0,Y 195.6,Z 516.157,A -85,B 0,C 180,E1 -25751.745,E2 -25751.745} C_VEL
LIN {X 0,Y 190.846,Z 529.038,A -85,B 0,C 180,E1 -25752.827,E2 -25752.827} C_VEL
LIN {X 0,Y 184.91,Z 541.89,A -85,B 0,C 180,E1 -25754.268,E2 -25754.268} C_VEL
LIN {X 0,Y 178.03,Z 554.031,A -85,B 0,C 180,E1 -25756.041,E2 -25756.041} C_VEL
LIN {X 0,Y 171.637,Z 563.524,A -85,B 0,C 180,E1 -25757.83,E2 -25757.83} C_VEL
LIN {X 0,Y 164.581,Z 572.641,A -85,B 0,C 180,E1 -25760.048,E2 -25760.048} C_VEL
LIN {X 0,Y 156.474,Z 581.751,A -85,B 0,C 180,E1 -25762.971,E2 -25762.971} C_VEL
LIN {X 0,Y 147.578,Z 590.307,A -85,B 0,C 180,E1 -25766.764,E2 -25766.764} C_VEL
LIN {X 0,Y 139.417,Z 597.08,A -85,B 0,C 180,E1 -25771.028,E2 -25771.028} C_VEL
LIN {X 0,Y 132.072,Z 602.355,A -85,B 0,C 180,E1 -25775.826,E2 -25775.826} C_VEL
LIN {X 0,Y 127.51,Z 605.249,A -85,B 0,C 180,E1 -25779.504,E2 -25779.504} C_VEL
LIN {X 0,Y 124.029,Z 607.172,A -85,B 0,C 180,E1 -25782.84,E2 -25782.84} C_VEL
LIN {X 0,Y 118.754,Z 609.544,A -85,B 0,C 180,E1 -25789.388,E2 -25789.388} C_VEL
LIN {X 0,Y 114.885,Z 610.497,A -85,B 0,C 180,E1 -25796.598,E2 -25796.598} C_VEL
LIN {X 0,Y 112.601,Z 609.985,A -85,B 0,C 180,E1 -25804.097,E2 -25804.097} C_VEL
LIN {X 0,Y 111.838,Z 608.028,A -85,B 0,C 180,E1 -25811.691,E2 -25811.691} C_VEL
LIN {X 0,Y 112.323,Z 604.598,A -85,B 0,C 180,E1 -25819.184,E2 -25819.184} C_VEL
LIN {X 0,Y 113.588,Z 600.802,A -85,B 0,C 180,E1 -25824.968,E2 -25824.968} C_VEL
LIN {X 0,Y 115.246,Z 596.516,A -85,B 0,C 180,E1 -25830.003,E2 -25830.003} C_VEL
LIN {X 0,Y 118.166,Z 590.009,A -85,B 0,C 180,E1 -25835.977,E2 -25835.977} C_VEL
LIN {X 0,Y 121.74,Z 582.78,A -85,B 0,C 180,E1 -25841.074,E2 -25841.074} C_VEL
LIN {X 0,Y 125.506,Z 574.966,A -85,B 0,C 180,E1 -25845.428,E2 -25845.428} C_VEL
LIN {X 0,Y 130.179,Z 565.067,A -85,B 0,C 180,E1 -25849.723,E2 -25849.723} C_VEL
LIN {X 0,Y 135.079,Z 554.045,A -85,B 0,C 180,E1 -25853.376,E2 -25853.376} C_VEL
LIN {X 0,Y 139.879,Z 541.818,A -85,B 0,C 180,E1 -25856.484,E2 -25856.484} C_VEL
LIN {X 0,Y 144.01,Z 529.696,A -85,B 0,C 180,E1 -25858.814,E2 -25858.814} C_VEL
LIN {X 0,Y 147.583,Z 516.933,A -85,B 0,C 180,E1 -25860.685,E2 -25860.685} C_VEL
LIN {X 0,Y 150.532,Z 503.218,A -85,B 0,C 180,E1 -25862.179,E2 -25862.179} C_VEL
LIN {X 0,Y 152.746,Z 489.153,A -85,B 0,C 180,E1 -25863.22,E2 -25863.22} C_VEL
LIN {X 0,Y 154.539,Z 470.204,A -85,B 0,C 180,E1 -25864.041,E2 -25864.041} C_VEL
LIN {X 0,Y 157.698,Z 429.575,A -85,B 0,C 180,E1 -25865.552,E2 -25865.552} C_VEL
LIN {X 0,Y 152.53,Z 418.326,A -85,B 0,C 180,E1 -25868.438,E2 -25868.438} C_VEL
LIN {X 0,Y 147.183,Z 408.147,A -85,B 0,C 180,E1 -25871.732,E2 -25871.732} C_VEL
LIN {X 0,Y 141.744,Z 399.174,A -85,B 0,C 180,E1 -25875.465,E2 -25875.465} C_VEL
LIN {X 0,Y 137.987,Z 393.798,A -85,B 0,C 180,E1 -25878.357,E2 -25878.357} C_VEL
LIN {X 0,Y 135.684,Z 390.534,A -85,B 0,C 180,E1 -25880.338,E2 -25880.338} C_VEL
LIN {X 0,Y 132.786,Z 386.481,A -85,B 0,C 180,E1 -25883.122,E2 -25883.122} C_VEL
LIN {X 0,Y 130.15,Z 383.027,A -85,B 0,C 180,E1 -25886.005,E2 -25886.005} C_VEL
LIN {X 0,Y 129.53,Z 381.929,A -85,B 0,C 180,E1 -25886.791,E2 -25886.791} C_VEL
LIN {X 0,Y 126.923,Z 379.491,A -85,B 0,C 180,E1 -25890.11,E2 -25890.11} C_VEL
LIN {X 0,Y 125.495,Z 376.717,A -85,B 0,C 180,E1 -25892.501,E2 -25892.501} C_VEL
LIN {X 0,Y 122.566,Z 374.664,A -85,B 0,C 180,E1 -25897.953,E2 -25897.953} C_VEL
LIN {X 0,Y 121.093,Z 371.685,A -85,B 0,C 180,E1 -25902.915,E2 -25902.915} C_VEL
LIN {X 0,Y 120.922,Z 370.877,A -85,B 0,C 180,E1 -25903.975,E2 -25903.975} C_VEL
LIN {X 0,Y 120.275,Z 370.628,A -85,B 0,C 180,E1 -25913.416,E2 -25913.416} C_VEL
LIN {X 0,Y 121.61,Z 370.855,A -85,B 0,C 180,E1 -25919.898,E2 -25919.898} C_VEL
LIN {X 0,Y 122.339,Z 373.506,A -85,B 0,C 180,E1 -25922.676,E2 -25922.676} C_VEL
LIN {X 0,Y 124.493,Z 375.944,A -85,B 0,C 180,E1 -25927.298,E2 -25927.298} C_VEL
LIN {X 0,Y 125.891,Z 376.861,A -85,B 0,C 180,E1 -25929.541,E2 -25929.541} C_VEL
LIN {X 0,Y 127.573,Z 379.968,A -85,B 0,C 180,E1 -25932.218,E2 -25932.218} C_VEL
LIN {X 0,Y 130.004,Z 382.385,A -85,B 0,C 180,E1 -25935.236,E2 -25935.236} C_VEL
LIN {X 0,Y 132.626,Z 386.116,A -85,B 0,C 180,E1 -25938.165,E2 -25938.165} C_VEL
LIN {X 0,Y 133.818,Z 387.776,A -85,B 0,C 180,E1 -25939.363,E2 -25939.363} C_VEL
LIN {X 0,Y 137.071,Z 392.33,A -85,B 0,C 180,E1 -25942.322,E2 -25942.322} C_VEL
LIN {X 0,Y 140.597,Z 397.458,A -85,B 0,C 180,E1 -25945.145,E2 -25945.145} C_VEL
LIN {X 0,Y 145.798,Z 405.727,A -85,B 0,C 180,E1 -25948.819,E2 -25948.819} C_VEL
LIN {X 0,Y 148.261,Z 410.683,A -85,B 0,C 180,E1 -25950.477,E2 -25950.477} C_VEL
LIN {X 0,Y 152.386,Z 421.033,A -85,B 0,C 180,E1 -25953.162,E2 -25953.162} C_VEL
LIN {X 0,Y 156.53,Z 433.275,A -85,B 0,C 180,E1 -25955.711,E2 -25955.711} C_VEL
LIN {X 0,Y 157.335,Z 436.049,A -85,B 0,C 180,E1 -25956.203,E2 -25956.203} C_VEL
LIN {X 0,Y 152.802,Z 493.835,A -85,B 0,C 180,E1 -25958.443,E2 -25958.443} C_VEL
LIN {X 0,Y 150.596,Z 508.369,A -85,B 0,C 180,E1 -25959.378,E2 -25959.378} C_VEL
LIN {X 0,Y 147.777,Z 521.897,A -85,B 0,C 180,E1 -25960.712,E2 -25960.712} C_VEL
LIN {X 0,Y 143.991,Z 535.032,A -85,B 0,C 180,E1 -25962.416,E2 -25962.416} C_VEL
LIN {X 0,Y 140.032,Z 546.923,A -85,B 0,C 180,E1 -25964.533,E2 -25964.533} C_VEL
LIN {X 0,Y 136.529,Z 556.313,A -85,B 0,C 180,E1 -25966.661,E2 -25966.661} C_VEL
LIN {X 0,Y 132.359,Z 566.149,A -85,B 0,C 180,E1 -25969.421,E2 -25969.421} C_VEL
LIN {X 0,Y 127.894,Z 575.685,A -85,B 0,C 180,E1 -25972.806,E2 -25972.806} C_VEL
LIN {X 0,Y 123.323,Z 585.283,A -85,B 0,C 180,E1 -25977.219,E2 -25977.219} C_VEL
LIN {X 0,Y 119.516,Z 593.219,A -85,B 0,C 180,E1 -25981.935,E2 -25981.935} C_VEL
LIN {X 0,Y 116.473,Z 599.783,A -85,B 0,C 180,E1 -25986.905,E2 -25986.905} C_VEL
LIN {X 0,Y 114.262,Z 605.198,A -85,B 0,C 180,E1 -25992.086,E2 -25992.086} C_VEL
LIN {X 0,Y 112.689,Z 610.875,A -85,B 0,C 180,E1 -25999.213,E2 -25999.213} C_VEL
LIN {X 0,Y 112.388,Z 613.091,A -85,B 0,C 180,E1 -26002.812,E2 -26002.812} C_VEL
LIN {X 0,Y 112.49,Z 616.355,A -85,B 0,C 180,E1 -26009.997,E2 -26009.997} C_VEL
LIN {X 0,Y 112.33,Z 617.405,A -85,B 0,C 180,E1 -26013.584,E2 -26013.584} C_VEL
LIN {X 0,Y 112.682,Z 618.492,A -85,B 0,C 180,E1 -26020.781,E2 -26020.781} C_VEL
LIN {X 0,Y 114.446,Z 618.288,A -85,B 0,C 180,E1 -26027.878,E2 -26027.878} C_VEL
LIN {X 0,Y 117.929,Z 616.809,A -85,B 0,C 180,E1 -26034.652,E2 -26034.652} C_VEL
LIN {X 0,Y 122.816,Z 614.023,A -85,B 0,C 180,E1 -26040.995,E2 -26040.995} C_VEL
LIN {X 0,Y 125.39,Z 612.414,A -85,B 0,C 180,E1 -26043.488,E2 -26043.488} C_VEL
LIN {X 0,Y 127.453,Z 610.804,A -85,B 0,C 180,E1 -26045.891,E2 -26045.891} C_VEL
LIN {X 0,Y 129.682,Z 607.797,A -85,B 0,C 180,E1 -26049.987,E2 -26049.987} C_VEL
LIN {X 0,Y 132.424,Z 604.212,A -85,B 0,C 180,E1 -26053.847,E2 -26053.847} C_VEL
LIN {X 0,Y 135.186,Z 601.698,A -85,B 0,C 180,E1 -26055.806,E2 -26055.806} C_VEL
LIN {X 0,Y 143.281,Z 595.045,A -85,B 0,C 180,E1 -26059.484,E2 -26059.484} C_VEL
LIN {X 0,Y 152.331,Z 586.399,A -85,B 0,C 180,E1 -26062.924,E2 -26062.924} C_VEL
LIN {X 0,Y 160.045,Z 577.918,A -85,B 0,C 180,E1 -26065.418,E2 -26065.418} C_VEL
LIN {X 0,Y 168.345,Z 567.4,A -85,B 0,C 180,E1 -26067.709,E2 -26067.709} C_VEL
LIN {X 0,Y 176.198,Z 555.669,A -85,B 0,C 180,E1 -26069.6,E2 -26069.6} C_VEL
LIN {X 0,Y 182.843,Z 543.911,A -85,B 0,C 180,E1 -26070.975,E2 -26070.975} C_VEL
LIN {X 0,Y 188.823,Z 530.985,A -85,B 0,C 180,E1 -26072.121,E2 -26072.121} C_VEL
LIN {X 0,Y 193.732,Z 517.486,A -85,B 0,C 180,E1 -26073,E2 -26073} C_VEL
LIN {X 0,Y 197.636,Z 502.996,A -85,B 0,C 180,E1 -26073.648,E2 -26073.648} C_VEL
LIN {X 0,Y 200.222,Z 488.099,A -85,B 0,C 180,E1 -26074.127,E2 -26074.127} C_VEL
LIN {X 0,Y 201.859,Z 473.183,A -85,B 0,C 180,E1 -26074.497,E2 -26074.497} C_VEL
LIN {X 0,Y 199.928,Z 466.914,A -85,B 0,C 180,E1 -26077.177,E2 -26077.177} C_VEL
LIN {X 0,Y 198.439,Z 462.66,A -85,B 0,C 180,E1 -26079.569,E2 -26079.569} C_VEL
LIN {X 0,Y 197.191,Z 458.995,A -85,B 0,C 180,E1 -26082.197,E2 -26082.197} C_VEL
LIN {X 0,Y 196.211,Z 456.282,A -85,B 0,C 180,E1 -26084.946,E2 -26084.946} C_VEL
LIN {X 0,Y 195.195,Z 454.013,A -85,B 0,C 180,E1 -26091.719,E2 -26091.719} C_VEL
LIN {X 0,Y 196.309,Z 455.942,A -85,B 0,C 180,E1 -26097.751,E2 -26097.751} C_VEL
LIN {X 0,Y 198.014,Z 460.057,A -85,B 0,C 180,E1 -26101.91,E2 -26101.91} C_VEL
LIN {X 0,Y 199.994,Z 464.372,A -85,B 0,C 180,E1 -26105.102,E2 -26105.102} C_VEL
LIN {X 0,Y 202.185,Z 469.338,A -85,B 0,C 180,E1 -26107.902,E2 -26107.902} C_VEL
LIN {X 0,Y 199.718,Z 489.924,A -85,B 0,C 180,E1 -26108.48,E2 -26108.48} C_VEL
LIN {X 0,Y 196.824,Z 503.702,A -85,B 0,C 180,E1 -26109.036,E2 -26109.036} C_VEL
LIN {X 0,Y 192.611,Z 517.895,A -85,B 0,C 180,E1 -26109.892,E2 -26109.892} C_VEL
LIN {X 0,Y 187.574,Z 530.853,A -85,B 0,C 180,E1 -26110.98,E2 -26110.98} C_VEL
LIN {X 0,Y 181.644,Z 543.078,A -85,B 0,C 180,E1 -26112.337,E2 -26112.337} C_VEL
LIN {X 0,Y 175.061,Z 554.263,A -85,B 0,C 180,E1 -26113.937,E2 -26113.937} C_VEL
LIN {X 0,Y 167.985,Z 564.413,A -85,B 0,C 180,E1 -26115.802,E2 -26115.802} C_VEL
LIN {X 0,Y 160.684,Z 573.44,A -85,B 0,C 180,E1 -26117.975,E2 -26117.975} C_VEL
LIN {X 0,Y 152.28,Z 582.437,A -85,B 0,C 180,E1 -26120.849,E2 -26120.849} C_VEL
LIN {X 0,Y 143.017,Z 590.889,A -85,B 0,C 180,E1 -26124.625,E2 -26124.625} C_VEL
LIN {X 0,Y 135.623,Z 596.741,A -85,B 0,C 180,E1 -26128.25,E2 -26128.25} C_VEL
LIN {X 0,Y 128.849,Z 601.463,A -85,B 0,C 180,E1 -26132.29,E2 -26132.29} C_VEL
LIN {X 0,Y 122.76,Z 605.113,A -85,B 0,C 180,E1 -26136.732,E2 -26136.732} C_VEL
LIN {X 0,Y 115.884,Z 608.564,A -85,B 0,C 180,E1 -26143.306,E2 -26143.306} C_VEL
LIN {X 0,Y 110.613,Z 610.397,A -85,B 0,C 180,E1 -26150.557,E2 -26150.557} C_VEL
LIN {X 0,Y 107.04,Z 610.739,A -85,B 0,C 180,E1 -26158.318,E2 -26158.318} C_VEL
LIN {X 0,Y 105.108,Z 609.626,A -85,B 0,C 180,E1 -26166.352,E2 -26166.352} C_VEL
LIN {X 0,Y 104.77,Z 608.527,A -85,B 0,C 180,E1 -26170.407,E2 -26170.407} C_VEL
LIN {X 0,Y 105.095,Z 605.249,A -85,B 0,C 180,E1 -26178.431,E2 -26178.431} C_VEL
LIN {X 0,Y 106.082,Z 602.24,A -85,B 0,C 180,E1 -26183.581,E2 -26183.581} C_VEL
LIN {X 0,Y 108.035,Z 597.391,A -85,B 0,C 180,E1 -26190.003,E2 -26190.003} C_VEL
LIN {X 0,Y 110.992,Z 591.035,A -85,B 0,C 180,E1 -26196.365,E2 -26196.365} C_VEL
LIN {X 0,Y 115.037,Z 583.326,A -85,B 0,C 180,E1 -26202.186,E2 -26202.186} C_VEL
LIN {X 0,Y 119.37,Z 574.834,A -85,B 0,C 180,E1 -26207.123,E2 -26207.123} C_VEL
LIN {X 0,Y 124.342,Z 564.853,A -85,B 0,C 180,E1 -26211.558,E2 -26211.558} C_VEL
LIN {X 0,Y 129.497,Z 553.741,A -85,B 0,C 180,E1 -26215.305,E2 -26215.305} C_VEL
LIN {X 0,Y 134.576,Z 541.336,A -85,B 0,C 180,E1 -26218.462,E2 -26218.462} C_VEL
LIN {X 0,Y 139.082,Z 528.419,A -85,B 0,C 180,E1 -26220.918,E2 -26220.918} C_VEL
LIN {X 0,Y 142.755,Z 515.389,A -85,B 0,C 180,E1 -26222.792,E2 -26222.792} C_VEL
LIN {X 0,Y 145.839,Z 501.124,A -85,B 0,C 180,E1 -26224.282,E2 -26224.282} C_VEL
LIN {X 0,Y 148.01,Z 487.11,A -85,B 0,C 180,E1 -26225.25,E2 -26225.25} C_VEL
LIN {X 0,Y 150.854,Z 454.822,A -85,B 0,C 180,E1 -26226.527,E2 -26226.527} C_VEL
LIN {X 0,Y 152.656,Z 431.993,A -85,B 0,C 180,E1 -26227.4,E2 -26227.4} C_VEL
LIN {X 0,Y 148.245,Z 422.137,A -85,B 0,C 180,E1 -26230.102,E2 -26230.102} C_VEL
LIN {X 0,Y 143.098,Z 412.178,A -85,B 0,C 180,E1 -26233.548,E2 -26233.548} C_VEL
LIN {X 0,Y 138.55,Z 404.486,A -85,B 0,C 180,E1 -26236.93,E2 -26236.93} C_VEL
LIN {X 0,Y 133.782,Z 397.231,A -85,B 0,C 180,E1 -26241.047,E2 -26241.047} C_VEL
